(* CODESYS project XPlanarApplication143.library
   Placeholder: XPlanarApplication
   Version: 1.4.3
   Title: XPlanarApplication
   DefaultNamespace: XPlanarApplication
   Company: Beckhoff Automation LLC

Project tree, tasks and I/O mapping:
  libraries: SPT Base Types, * (Beckhoff Automation LLC); Tc2_Math, * (Beckhoff Automation GmbH); Tc2_Standard, * (Beckhoff Automation GmbH); Tc2_System, * (Beckhoff Automation GmbH); Tc2_Utilities, * (Beckhoff Automation GmbH); Tc3_EventLogger, * (Beckhoff Automation GmbH); Tc3_Mc3PlanarMotion, * (Beckhoff Automation GmbH); Tc3_Module, * (Beckhoff Automation GmbH); Tc3_Physics, * (Beckhoff Automation GmbH); Tc3_XPlanarUtility, * (Beckhoff Automation GmbH)
  Mover/
    DUTs/
      data type ST_CommandLog
      data type ST_MoveDynamics
      data type ST_MoverCommand
      data type ST_MoverHMI
      data type ST_MoverObjectInfos
    TaskClasses/
      function block FB_AddToGroup [ST]: Execute
      function block FB_Disable [ST]: Execute
      function block FB_Enable [ST]: Execute
      function block FB_EnterMovementArea [ST]: Execute, Update
      function block FB_Halt [ST]: Execute
      function block FB_JoinClosestTrack [ST]: Execute, Update
      function block FB_JoinTrack [ST]: Execute
      function block FB_LeaveMovementArea [ST]: Execute, Update
      function block FB_LeaveTrack [ST]: Execute
      function block FB_MoveA [ST]: Execute
      function block FB_MoveB [ST]: Execute
      function block FB_MoveToPosition [ST]: Execute
      function block FB_MoveZ [ST]: Execute
      function block FB_ResetMover [ST]: Execute
      function block FB_Rotate [ST]: Execute
      function block FB_RunExternalSetpointAbsoluteMode [ST]: Execute
      function block FB_RunExternalSetpointRelativeMode [ST]: Execute
      function block FB_SquareUp [ST]: Execute, Update
      function block FB_StopExternalSetpoint [ST]: Execute
      function block FB_TrackMove [ST]: Execute
      function block FB_TrackMoveXY [ST]: Execute
    function block FB_XPlanarMover [ST]: FreeMove, JoinClosestTrack, JoinTrack, LeaveTrack, Rotate, RunExternalSpAbsoluteMode, RunExternalSpRelativeMode, SendToStation, SquareUp, StopExternalSp, TiltA, TiltB, TrackMove, TrackMoveXY, VerticalMove, Movement, Rotation, Tilt, ActualPosition, AddToGroup, AtRotationPosition, CommandLog, Destination, Disable, Dynamics, Enable, EnterMovementArea, Gap, Halt, IdentifiedBTN, InStation, LeaveMovementArea, MoveCommand, MoverBTN, MoverIndex, MoverType, pm, Reset, RotationModulo, Status, Utility, CyclicLogic, Initialize
    interface I_MoveCommands: FreeMove, JoinClosestTrack, JoinTrack, LeaveTrack, Rotate, RunExternalSpAbsoluteMode, RunExternalSpRelativeMode, SendToStation, SquareUp, StopExternalSp, TiltA, TiltB, TrackMove, TrackMoveXY, VerticalMove
    interface I_MoveDynamics: Movement, Rotation, Tilt
    interface I_XPlanarMover: ActualPosition, AddToGroup, AtRotationPosition, CommandLog, CyclicLogic, Destination, Disable, Dynamics, Enable, EnterMovementArea, Gap, Halt, IdentifiedBTN, InStation, LeaveMovementArea, MoveCommand, MoverBTN, MoverIndex, MoverType, pm, Reset, RotationModulo, Status, Utility
  Part/
    Tasks/
      function block FB_AllowEnable [ST]: Execute
      function block FB_ForceDisable [ST]: Execute
      function block FB_Initialize [ST]: Execute
      function block FB_ResetPart [ST]: Execute
    function block FB_XPlanarPart [ST]: CyclicLogic, ForceDisable, Initialize, ObjectID, pm, Reset, SetAllowEnable, State
    interface I_XPlanarPart: ForceDisable, ObjectID, pm, Reset, SetAllowEnable, State
  Station/
    DUT/
      data type E_StationType
      data type E_XplanarStationState
      data type ST_StationHMI
      data type ST_XPlanarStationObjectInfos
    function block FB_MoverQueue [ST]: Clear, Count, Dequeue, Enqueue, FirstMover, LastMover, MoverIDs, Queue
    function block FB_XPlanarStationBase [ST]: AllowQueing, CanReleaseMover, CurrentMover, Error, Execute, HasMover, ID, MoverQueue, NextStation, NumMoversRequired, Position, Reset, Size, StationComplete, StationReady, StationType, TrackID, CyclicLogic, Name, WatchForMover
    interface I_XPlanarStation: AllowQueing, CanReleaseMover, CurrentMover, Execute, HasMover, ID, MoverQueue, Name, NextStation, NumMoversRequired, Position, Reset, Size, StationComplete, StationReady, StationType, TrackID
  Tile/
    DUT/
      data type ST_TileObjectInfos
      data type ST_TileTemperatures
    function block FB_XPlanarTile [ST]: Btn, CyclicLogic, DcLinkOk, Index, Initialize, PartIndex, PositionOnPart, Temperatures, TimeToShutdown, Update, Utility
    interface I_XPlanarTile: Btn, DcLinkOk, Index, PartIndex, PositionOnPart, Temperatures, TimeToShutdown, Update, Utility
  Track/
    DUT/
      data type E_TrackItemType
      data type ST_TrackDefinition
      data type ST_TrackItems
      data type ST_TrackStatus
    TaskClasses/
      function block FB_AddTrackToGroup [ST]: Execute
      function block FB_AppendLine [ST]: Execute
      function block FB_AppendPoint [ST]: Execute
      function block FB_BuildTrack [ST]: Execute, Update
      function block FB_ClearSegment [ST]: Execute
      function block FB_CloseLoop [ST]: Execute
      function block FB_DisableTrack [ST]: Execute
      function block FB_EnableTrack [ST]: Execute
      function block FB_SetEndAtTrack [ST]: Execute
      function block FB_SetStartFromTrack [ST]: Execute
      function block FB_TrackReset [ST]: Execute
    function block FB_XPlanarTrackSegment [ST]: AddToGroup, AppendLine, AppendPoint, Build, Clear, CloseLoop, Definition, Disable, Enable, GetTrackPositionAt, Index, IsStanding, MoverCount, MovingMoverCount, pm, Reset, SetEndAtTrack, SetStartFromTrack, Status, TrackLength, Utility, CyclicLogic
    interface I_XPlanarTrack: AddToGroup, AppendLine, AppendPoint, Build, Clear, CloseLoop, CyclicLogic, Definition, Disable, Enable, GetTrackPositionAt, Index, MoverCount, MovingMoverCount, pm, Reset, Status, TrackLength, Utility
  XPlanarComponent/
    TaskClasses/
      function block FB_EnableGroup [ST]: Execute
      function block FB_MoverIdentification [ST]: Execute, Update
      function block FB_MoverRedetection [ST]: Execute, MoverDetectionInfo, Update
      function block FB_ResetGroup [ST]: Execute
      function block FB_ResetXPlanar [ST]: Execute, Update
    function block FB_Component_XPlanar [ST]: Monitoring, CyclicLogic, Abort, AddMoversToGroup, AddTracksToGroup, DisableMovers, EnableGroup, EnableMovers, EnableTracks, IdentifyMovers, Initialize, MoverDetectionInfo, MoverRedetect, Reset, TileCount, TracksInitialized, Utility
  XPlanarResultClasses/
    function block FB_MoverTaskResult [ST]: Mover, Update, UpdateLog
    function block FB_PartTaskResult [ST]: Part
    function block FB_PlanarFeedbackResult [ST]: PlanarFeedback, Update
    function block FB_ResultBase [ST]: Aborted, BlockingObjectInfo, Busy, Done, Error, ErrorID, Result, TaskName
    function block FB_TrackTaskResult [ST]: Track
    interface I_PlanarTaskResult: Aborted, BlockingObjectInfo, Busy, Done, Error, ErrorID
  global variables ip
  00000000-0000-0000-0000-000000000000|LICENSE
  LICENSE
  global variables SystemParameters
  global variables XPlanar
  global variables XPlanarHMI
*)

// Mover/DUTs/ST_CommandLog
TYPE ST_CommandLog EXTENDS ST_MoverCommand :
	STRUCT
		Timestamp : STRING(24);
	END_STRUCT
END_TYPE

// Mover/DUTs/ST_MoveDynamics
TYPE ST_MoveDynamics :
STRUCT
	Velocity	: LREAL;
	Accel		: LREAL;
	Decel		: LREAL;
	Jerk		: LREAL;
END_STRUCT
END_TYPE

// Mover/DUTs/ST_MoverCommand
TYPE ST_MoverCommand :
	STRUCT
		Command : STRING;
		Vlocity : LREAL;
		Accel	: LREAL;
		Decel	: LREAL;
		Jerk	: LREAL;
	END_STRUCT
END_TYPE

// Mover/DUTs/ST_MoverHMI
TYPE ST_MoverHMI :
	STRUCT
		Enabled		   : BOOL;
		Error		   : BOOL;
		InStation	   : BOOL;
		ErrorID		   : UDINT;
		CurrentStation : STRING;
		CommandMode	   : STRING;
		LastCommand	   : STRING;
		EnableMover	   : BOOL;
		DisableMover   : BOOL;
		ResetMover	   : BOOL;
		HaltMover	   : BOOL;
	END_STRUCT
END_TYPE

// Mover/DUTs/ST_MoverObjectInfos
TYPE ST_MoverObjectInfos :
	STRUCT
		Width	 : DINT;
		Height	 : DINT;
		MoverBTN : STRING(13);
	END_STRUCT
END_TYPE

// Station/DUT/E_StationType
{attribute 'qualified_only'}
TYPE E_StationType : (
		Process		  := 0,
		DecisionPoint := 1,
		MultiMover	  := 2
	) UDINT;
END_TYPE

// Station/DUT/E_XplanarStationState
{attribute 'qualified_only'}
{attribute 'strict'}
{attribute 'to_string'}
TYPE E_XplanarStationState : (
		StationIdle := 0,
		ProcessMover,
		SquareUpMover,
		SendMoverAway,
		CycleComplete,
		SendQueue,
		StationError
	);
END_TYPE

// Station/DUT/ST_StationHMI
TYPE ST_StationHMI :
	STRUCT
		Error		   : BOOL;
		Reset		   : BOOL;
		StationReady   : BOOL;
		HasMover	   : BOOL;
		CurrentMoverID : STRING(13);
		CurrentState   : STRING;
	END_STRUCT
END_TYPE

// Station/DUT/ST_XPlanarStationObjectInfos
TYPE ST_XPlanarStationObjectInfos :
	STRUCT
		X	   : DINT;
		Y	   : DINT;
		Width  : DINT;
		Height : DINT;
	END_STRUCT
END_TYPE

// Tile/DUT/ST_TileObjectInfos
TYPE ST_TileObjectInfos :
	STRUCT
		X	   : DINT;
		Y	   : DINT;
		Width  : DINT;
		Height : DINT;
	END_STRUCT
END_TYPE

// Tile/DUT/ST_TileTemperatures
TYPE ST_TileTemperatures :
	STRUCT
		Center : LREAL;
		East   : LREAL;
		West   : LREAL;
		North  : LREAL;
		South  : LREAL;
	END_STRUCT
END_TYPE

// Track/DUT/E_TrackItemType
TYPE E_TrackItemType :
(
	Point := 0,
	Line,
	Circle
);
END_TYPE

// Track/DUT/ST_TrackDefinition
TYPE ST_TrackDefinition :
	STRUCT
		StartFromTrackID : UDINT;
		EndAtTrackID	 : UDINT;
		CloseLoop		 : BOOL;
		Items			 : ARRAY[1..SystemParameters.MAX_OBJECTS_PER_TRACK] OF ST_TrackItems;
	END_STRUCT
END_TYPE

// Track/DUT/ST_TrackItems
TYPE ST_TrackItems :
STRUCT
	ItemType		: E_TrackItemType;
	StartPoint		: PositionXYC;
	EndPoint		: PositionXYC;
	CenterPoint		: PositionXY;
	CircleClockwise : BOOL;
END_STRUCT
END_TYPE

// Track/DUT/ST_TrackStatus
TYPE ST_TrackStatus :
	STRUCT
		State			 : MC_PLANAR_STATE;
		OperationMode	 : MC_PLANAR_TRACK_OPERATION_MODE;
		MoverCount		 : UDINT;
		CalculatedLength : LREAL;
	END_STRUCT
END_TYPE

// ip
{attribute 'qualified_only'}
VAR_GLOBAL
	Movers	 : ARRAY[0..SystemParameters.MOVER_COUNT] OF I_XPlanarMover;
	Tracks	 : ARRAY[0..SystemParameters.TRACK_COUNT] OF I_XPlanarTrack;
	Stations : ARRAY[0..SystemParameters.STATION_COUNT] OF I_XPlanarStation;
END_VAR

// SystemParameters
{attribute 'qualified_only'}
VAR_GLOBAL CONSTANT
	EnableCommandTracing  : BOOL  := FALSE; //Enables mover command trace logging
	AssumedMoverSize	  : LREAL := 50;
	MAX_LOG_COUNT		  : UINT  := 20; //Size of command mover log
	MOVER_COUNT			  : UINT  := 1;	 //Total number of movers configured in the system
	TRACK_COUNT			  : UINT  := 1;	 //Total number of track segments in the system
	MAX_OBJECTS_PER_TRACK : UINT  := 20; //Maximum number of points or lines defined in a single track segment
	STATION_COUNT		  : UINT  := 3;	 //Total number of stations in the system
	MaxMoversPerStation	  : UDINT := 4;	 //Max number of movers allowed to queue in a station 
	TileDiagUpdate		  : LREAL := 0;	 //Tile Diagnostic data update rate in seconds.  Set to 0 to disable
END_VAR

// XPlanar
{attribute 'qualified_only'}
VAR_GLOBAL
	Environment		   : Tc3_MC3PlanarMotion.MC_PlanarEnvironment;
	EnvironmentTcIo	   : Tc3_XPlanarUtility.FB_TcIoXPlanarEnvironment;
	Group			   : Tc3_MC3PlanarMotion.MC_PlanarGroup;
	Parts			   : ARRAY[1..Param_TcIoXPlanarEnvironment.MaxParts] OF FB_XPlanarPart;
	Tiles			   : ARRAY[1..Param_TcIoXPlanarEnvironment.MaxTiles] OF FB_XPlanarTile;
	OperationMode	   : XPlanarOperationMode;
	RotationMultiplier : LREAL := 120.0;
	XPUCount		   : UINT;
	PartCount		   : UINT;
	TrackCount		   : UINT;
	MoverCount		   : UINT;
	TileCount		   : UINT;
END_VAR

// XPlanarHMI
{attribute 'qualified_only'}
VAR_GLOBAL
	MoverObjects	: ARRAY[1..SystemParameters.MOVER_COUNT] OF ST_MoverObjectInfos;
	MoverPositions	: ARRAY[1..SystemParameters.MOVER_COUNT] OF MoverVector;
	TileObjects		: ARRAY[1..Param_TcIoXPlanarEnvironment.MaxTiles] OF ST_TileObjectInfos;
	StationObjects	: ARRAY[1..SystemParameters.STATION_COUNT] OF ST_XPlanarStationObjectInfos;
END_VAR

// Mover/TaskClasses/FB_AddToGroup
FUNCTION_BLOCK FB_AddToGroup EXTENDS FB_MoverTaskResult
VAR
END_VAR

METHOD Execute : I_PlanarTaskResult
VAR_INPUT
	Group : REFERENCE TO MC_PlanarGroup;
END_VAR
IF NOT HasRun THEN
	_Done	 := FALSE;
	_Error	 := FALSE;
	_Busy	 := FALSE;
	_ErrorID := 0;
	ipMover.pm.AddToGroup(_PlanarFb, Group);

	//Update mover command log				
	LogEntry.Command := CONCAT('AddMoverToGroup ', TO_STRING(Group.MCTOPLC_STD.GroupOID));
	LogEntry.Accel	 := 0;
	LogEntry.Decel	 := 0;
	LogEntry.Jerk	 := 0;
	LogEntry.Vlocity := 0;
	UpdateLog();
	HasRun := TRUE;
END_IF

Execute := THIS^;

//Heartbeat that the method is active
ExecuteWatchdog := ExecuteWatchdog + 1;
END_METHOD

END_FUNCTION_BLOCK

// XPlanarResultClasses/FB_MoverTaskResult
{attribute 'no_explicit_call' := 'do not call this POU directly'}
FUNCTION_BLOCK FB_MoverTaskResult EXTENDS FB_PlanarFeedbackResult
VAR
	ipMover : I_XPlanarMover;

	//CmdLog		   : REFERENCE TO ARRAY[0..SystemParameters.MAX_LOG_COUNT] OF ST_CommandLog;
	GetTime		   : GETSYSTEMTIME;
	SysTime		   : T_FILETIME;
	LogEntry	   : ST_MoverCommand;
	ActualPosition : MoverVector;
	RT_ADSWarn	   : R_Trig;
	MoverStr	   : STRING;
END_VAR

PROPERTY Mover : I_XPlanarMover
SET
ipMover := Mover;
END_SET
END_PROPERTY

METHOD Update
ActualPosition := ipMover.ActualPosition;
SUPER^.Update();
RT_ADSWarn(CLK := _PlanarFb.Error);
IF RT_ADSWarn.Q THEN
	MoverStr := CONCAT('Mover ', TO_STRING(ipMover.MoverIndex));
	LogEntry.Command := CONCAT(CONCAT(MoverStr, ' : %s'), CONCAT(LogEntry.Command, CONCAT('Error ', TO_STRING(_PlanarFb.ErrorId))));
	UpdateLog();
END_IF
END_METHOD

METHOD UpdateLog
VAR_INST
	i : UINT;
END_VAR
IF SystemParameters.MAX_LOG_COUNT > 0 THEN
	FOR i := SystemParameters.MAX_LOG_COUNT - 1 TO 1 BY -1 DO
		IF i < SystemParameters.MAX_LOG_COUNT THEN
			ipMover.CommandLog[i + 1] := ipMover.CommandLog[i];
		END_IF
	END_FOR

	ipMover.CommandLog[1] := ipMover.CommandLog[0];
	GetTime(timeLoDW => SysTime.dwLowDateTime, timeHiDW => SysTime.dwHighDateTime);
	ipMover.CommandLog[0].Timestamp := SYSTEMTIME_TO_STRING(FILETIME_TO_SYSTEMTIME(SysTime));
	ipMover.CommandLog[0].Command	:= LogEntry.Command;
	ipMover.CommandLog[0].Accel		:= LogEntry.Accel;
	ipMover.CommandLog[0].Decel		:= LogEntry.Decel;
	ipMover.CommandLog[0].Jerk		:= LogEntry.Jerk;
	ipMover.CommandLog[0].Vlocity	:= LogEntry.Vlocity;
END_IF
END_METHOD

END_FUNCTION_BLOCK

// XPlanarResultClasses/FB_PlanarFeedbackResult
{attribute 'no_assign_warning'}
{attribute 'no_explicit_call' := 'do not call this POU directly'}
FUNCTION_BLOCK FB_PlanarFeedbackResult EXTENDS FB_ResultBase
VAR
	_PlanarFb		: MC_PlanarFeedback;
	HasRun			: BOOL;
	ExecuteWatchdog : UDINT;
	TaskState		: UDINT;
END_VAR

{attribute 'suppress_wrn_C0410'}
PROPERTY PlanarFeedback : REFERENCE TO MC_PlanarFeedback
GET
PlanarFeedback ref= _PlanarFb;
END_GET
END_PROPERTY

METHOD Update
VAR_INST
	WatchdogCheck : UDINT;
END_VAR
//Update Command Feedback Status
_PlanarFb.Update();

//Update Interface based on Command Feedback status
_Aborted			:= _PlanarFb.Aborted;
_Busy				:= _PlanarFb.Active OR _PlanarFb.Busy;
_Done				:= _PlanarFb.Done;
_Error				:= _PlanarFb.Error;
_ErrorID			:= _PlanarFb.ErrorId;
_BlockingObjectInfo := _PlanarFb.objectInfo;

//Heartbeat to know execute is active
IF ExecuteWatchdog <> WatchdogCheck THEN
	WatchdogCheck := ExecuteWatchdog;
ELSE
	HasRun			:= FALSE;
	ExecuteWatchdog := 0;
END_IF
END_METHOD

END_FUNCTION_BLOCK

// XPlanarResultClasses/FB_ResultBase
{attribute 'no_explicit_call' := 'do not call this POU directly'}
FUNCTION_BLOCK FB_ResultBase EXTENDS FB_BaseFB IMPLEMENTS I_PlanarTaskResult
VAR
	_TaskName			: STRING;
	_Done				: BOOL;
	_Aborted			: BOOL;
	_BlockingObjectInfo : PlanarObjectInfo;
END_VAR

{attribute 'monitoring' := 'call'}
PROPERTY Aborted : BOOL
GET
Aborted := _Aborted;
END_GET
SET
_Aborted := Aborted;
END_SET
END_PROPERTY

{attribute 'suppress_wrn_C0410'}
PROPERTY BlockingObjectInfo : REFERENCE TO Tc3_Mc3PlanarMotion.PlanarObjectInfo
GET
BlockingObjectInfo ref= _BlockingObjectInfo;
END_GET
END_PROPERTY

{attribute 'monitoring' := 'call'}
PROPERTY Busy : BOOL
GET
Busy := _Busy;
END_GET
SET
_Busy := Busy;
END_SET
END_PROPERTY

{attribute 'monitoring' := 'call'}
PROPERTY Done : BOOL
GET
Done := _Done;
END_GET
SET
_Done := Done;
END_SET
END_PROPERTY

{attribute 'monitoring' := 'call'}
PROPERTY Error : BOOL
GET
Error := _Error;
END_GET
SET
_Error := Error;
END_SET
END_PROPERTY

{attribute 'monitoring' := 'call'}
PROPERTY ErrorID : UDINT
GET
ErrorID := _ErrorID;
END_GET
SET
_ErrorID := ErrorID;
END_SET
END_PROPERTY

PROPERTY Result : I_PlanarTaskResult
GET
Result := THIS^;
END_GET
END_PROPERTY

PROPERTY TaskName : STRING
GET
TaskName := _TaskName;
END_GET
SET
_TaskName := TaskName;
END_SET
END_PROPERTY

END_FUNCTION_BLOCK

// XPlanarResultClasses/I_PlanarTaskResult
INTERFACE I_PlanarTaskResult

{attribute 'monitoring' := 'call'}
PROPERTY Aborted : BOOL
GET
END_GET
END_PROPERTY

{attribute 'suppress_wrn_C0410'}
PROPERTY BlockingObjectInfo : REFERENCE TO PlanarObjectInfo
GET
END_GET
END_PROPERTY

{attribute 'monitoring' := 'call'}
PROPERTY Busy : BOOL
GET
END_GET
END_PROPERTY

{attribute 'monitoring' := 'call'}
PROPERTY Done : BOOL
GET
END_GET
END_PROPERTY

{attribute 'monitoring' := 'call'}
PROPERTY Error : BOOL
GET
END_GET
END_PROPERTY

{attribute 'monitoring' := 'call'}
PROPERTY ErrorID : UDINT
GET
END_GET
END_PROPERTY

END_INTERFACE

// Mover/I_XPlanarMover
INTERFACE I_XPlanarMover EXTENDS I_BaseFb

{attribute 'suppress_wrn_C0410'}
PROPERTY ActualPosition : REFERENCE TO MoverVector
GET
END_GET
END_PROPERTY

METHOD AddToGroup : I_PlanarTaskResult
VAR_INPUT
	PlanarGroup : REFERENCE TO MC_PlanarGroup;
END_VAR
END_METHOD

PROPERTY AtRotationPosition : BOOL
GET
END_GET
END_PROPERTY

{attribute 'suppress_wrn_C0410'}
PROPERTY CommandLog : REFERENCE TO ARRAY [0..SystemParameters.MAX_LOG_COUNT] of ST_CommandLog
GET
END_GET
END_PROPERTY

{attribute 'hide'}
METHOD CyclicLogic
END_METHOD

PROPERTY Destination : I_XPlanarStation
GET
END_GET
SET
END_SET
END_PROPERTY

METHOD Disable : I_PlanarTaskResult
END_METHOD

PROPERTY Dynamics : I_MoveDynamics
GET
END_GET
END_PROPERTY

METHOD Enable : I_PlanarTaskResult
END_METHOD

METHOD EnterMovementArea : I_PlanarTaskResult
VAR_INPUT
	PartId		: OTCID;
	PositionX	: LREAL;
	PositionY	: LREAL;
END_VAR
END_METHOD

PROPERTY Gap : LREAL
GET
END_GET
SET
END_SET
END_PROPERTY

METHOD Halt : I_PlanarTaskResult
END_METHOD

PROPERTY IdentifiedBTN : STRING
GET
END_GET
SET
END_SET
END_PROPERTY

PROPERTY InStation : BOOL
GET
END_GET
SET
END_SET
END_PROPERTY

METHOD LeaveMovementArea : I_PlanarTaskResult
END_METHOD

PROPERTY MoveCommand : I_MoveCommands
GET
END_GET
END_PROPERTY

PROPERTY MoverBTN : STRING
GET
END_GET
END_PROPERTY

PROPERTY MoverIndex : UDINT
GET
END_GET
SET
END_SET
END_PROPERTY

PROPERTY MoverType : XplanarMoverType
GET
END_GET
SET
END_SET
END_PROPERTY

{attribute 'suppress_wrn_C0410'}
PROPERTY pm : REFERENCE TO MC_PlanarMover
GET
END_GET
END_PROPERTY

//! @summary Clears error flags and error IDs for this component
{attribute 'TcRpcEnable'}
METHOD PUBLIC Reset : I_PlanarTaskResult
END_METHOD

PROPERTY RotationModulo : LREAL
GET
END_GET
END_PROPERTY

{attribute 'suppress_wrn_C0410'}
PROPERTY Status : REFERENCE TO CDT_MCTOPLC_PLANAR_MOVER_STD
GET
END_GET
END_PROPERTY

PROPERTY Utility : I_TcIoXPlanarMover
GET
END_GET
SET
END_SET
END_PROPERTY

END_INTERFACE

// Station/I_XPlanarStation
INTERFACE I_XPlanarStation EXTENDS I_BaseFb

PROPERTY AllowQueing : BOOL
GET
END_GET
SET
END_SET
END_PROPERTY

PROPERTY CanReleaseMover : BOOL
SET
END_SET
END_PROPERTY

PROPERTY CurrentMover : I_XPlanarMover
GET
END_GET
END_PROPERTY

METHOD Execute
END_METHOD

PROPERTY HasMover : BOOL
GET
END_GET
SET
END_SET
END_PROPERTY

PROPERTY ID : UDINT
GET
END_GET
SET
END_SET
END_PROPERTY

{attribute 'suppress_wrn_C0410'}
PROPERTY MoverQueue : REFERENCE TO FB_MoverQueue
GET
END_GET
END_PROPERTY

PROPERTY Name : STRING
GET
END_GET
SET
END_SET
END_PROPERTY

PROPERTY NextStation : I_XPlanarStation
GET
END_GET
SET
END_SET
END_PROPERTY

PROPERTY NumMoversRequired : UDINT
GET
END_GET
SET
END_SET
END_PROPERTY

{attribute 'suppress_wrn_C0410'}
PROPERTY Position : REFERENCE TO PositionXYC
GET
END_GET
END_PROPERTY

METHOD Reset : BOOL
END_METHOD

{attribute 'suppress_wrn_C0410'}
PROPERTY Size : REFERENCE TO Position2D_LREAL
GET
END_GET
END_PROPERTY

PROPERTY StationComplete : BOOL
SET
END_SET
END_PROPERTY

PROPERTY StationReady : BOOL
GET
END_GET
END_PROPERTY

PROPERTY StationType : E_StationType
GET
END_GET
SET
END_SET
END_PROPERTY

PROPERTY TrackID : UDINT
GET
END_GET
SET
END_SET
END_PROPERTY

END_INTERFACE

// Station/FB_MoverQueue
//=============================================================================
//	FB_MoverQueue
//=============================================================================
//
//	FIFO Queue for use by stations
//
//-----------------------------------------------------------------------------

FUNCTION_BLOCK FB_MoverQueue
VAR
	MoversInQueue : UDINT := 0;
	ipMovers	  : ARRAY[1..SystemParameters.MaxMoversPerStation] OF I_XPlanarMover;
END_VAR

//=============================================================================
//	Method Clear()
//=============================================================================
//
//	Brute force reset of buffer
//
//-----------------------------------------------------------------------------
METHOD Clear : BOOL
MEMSET(ADR(ipMovers), 0, SIZEOF(ipMovers));
MoversInQueue := 0;
Clear		  := TRUE;
END_METHOD

PROPERTY Count : UDINT
GET
VAR
	i	 : UDINT;
	temp : UDINT;
END_VAR
Count := MoversInQueue;
END_GET
END_PROPERTY

METHOD Dequeue : BOOL
IF MoversInQueue > 0 THEN
	ipMovers[1].InStation := FALSE;
	MEMSET(ADR(ipMovers[1]), 0, SIZEOF(ipMovers[1]));
	MoversInQueue := MoversInQueue - 1;
	IF MoversInQueue > 0 THEN
		MEMMOVE(ADR(ipMovers[1]), ADR(ipMovers[2]), SIZEOF(ipMovers[2]) * MoversInQueue);
		MEMSET(ADR(ipMovers[MoversInQueue + 1]), 0, (SIZEOF(ipMovers[1]) * (SystemParameters.MaxMoversPerStation - MoversInQueue)));
	END_IF

	Dequeue := TRUE;
END_IF
END_METHOD

METHOD Enqueue : BOOL
VAR_INPUT
	ipMover : I_XPlanarMover;
END_VAR
IF MoversInQueue < SystemParameters.MaxMoversPerStation THEN
	MoversInQueue			:= MoversInQueue + 1;
	ipMover.InStation		:= TRUE;
	ipMovers[MoversInQueue] := ipMover;
	Enqueue					:= TRUE;
END_IF
END_METHOD

PROPERTY FirstMover : I_XPlanarMover
GET
IF MoversInQueue > 0 THEN
	FirstMover := ipMovers[1];
END_IF
END_GET
END_PROPERTY

PROPERTY LastMover : I_XPlanarMover
GET
IF MoversInQueue > 0 THEN
	LastMover := ipMovers[MoversInQueue];
END_IF
END_GET
END_PROPERTY

PROPERTY MoverIDs : ARRAY[1..SystemParameters.MaxMoversPerStation] OF UDINT
GET
VAR
	i : UDINT;
END_VAR
FOR i := 1 TO MoversInQueue DO
	IF ipMovers[i] <> 0 THEN
		MoverIDs[i] := ipMovers[i].MoverIndex;
	END_IF
END_FOR
END_GET
END_PROPERTY

{attribute 'suppress_wrn_C0410'}
PROPERTY Queue : REFERENCE TO ARRAY[1..SystemParameters.MaxMoversPerStation] OF I_XPlanarMover;
GET
VAR
	i : UDINT;
END_VAR
Queue ref= ipMovers;
END_GET
END_PROPERTY

END_FUNCTION_BLOCK

// Mover/I_MoveDynamics
INTERFACE I_MoveDynamics EXTENDS __SYSTEM.IQueryInterface

{attribute 'suppress_wrn_C0410'}
PROPERTY Movement : REFERENCE TO ST_MoveDynamics
GET
END_GET
END_PROPERTY

{attribute 'suppress_wrn_C0410'}
PROPERTY Rotation : REFERENCE TO ST_MoveDynamics
GET
END_GET
END_PROPERTY

{attribute 'suppress_wrn_C0410'}
PROPERTY Tilt : REFERENCE TO ST_MoveDynamics
GET
END_GET
END_PROPERTY

END_INTERFACE

// Mover/I_MoveCommands
INTERFACE I_MoveCommands EXTENDS __SYSTEM.IQueryInterface

METHOD FreeMove : I_PlanarTaskResult
VAR_INPUT
	XPosition : LREAL;
	YPosition : LREAL;
END_VAR
END_METHOD

{attribute 'TcRpcEnable'}
METHOD JoinClosestTrack : I_PlanarTaskResult
VAR_INPUT
	UseOrientation : BOOL;
END_VAR
END_METHOD

{attribute 'TcRpcEnable'}
METHOD JoinTrack : I_PlanarTaskResult
VAR_INPUT
	ipTrack		   : I_XPlanarTrack;
	UseOrientation : BOOL;
END_VAR
END_METHOD

{attribute 'TcRpcEnable'}
METHOD LeaveTrack : I_PlanarTaskResult
VAR_INPUT
	DestinationX   : LREAL;
	DestinationY   : LREAL;
	UseOrientation : BOOL;
END_VAR
END_METHOD

{attribute 'TcRpcEnable'}
METHOD Rotate : I_PlanarTaskResult
VAR_INPUT
	Position		: LREAL;
	AdditionalTurns : DINT;
END_VAR
END_METHOD

METHOD RunExternalSpAbsoluteMode : I_PlanarTaskResult
VAR_INPUT
	Position	 : MoverVector;
	Velocity	 : MoverVector;
	Acceleration : MoverVector;
END_VAR
END_METHOD

METHOD RunExternalSpRelativeMode : I_PlanarTaskResult
VAR_INPUT
	Position	 : MoverVector;
	Velocity	 : MoverVector;
	Acceleration : MoverVector;
END_VAR
END_METHOD

{attribute 'TcRpcEnable'}
METHOD SendToStation : I_PlanarTaskResult
VAR_INPUT
	Destination : I_XPlanarStation;
END_VAR
END_METHOD

{attribute 'TcRpcEnable'}
METHOD SquareUp : I_PlanarTaskResult
END_METHOD

METHOD StopExternalSp : I_PlanarTaskResult
END_METHOD

METHOD TiltA : I_PlanarTaskResult
VAR_INPUT
	Position : LREAL;
END_VAR
END_METHOD

METHOD TiltB : I_PlanarTaskResult
VAR_INPUT
	Position : LREAL;
END_VAR
END_METHOD

{attribute 'TcRpcEnable'}
METHOD TrackMove : I_PlanarTaskResult
VAR_INPUT
	Position : LREAL;
	Gap		  : LREAL;
	Track	  : I_XPlanarTrack;
	Direction : Tc3_Mc3PlanarMotion.MC_DIRECTION;
END_VAR
END_METHOD

{attribute 'TcRpcEnable'}
METHOD TrackMoveXY : I_PlanarTaskResult
VAR_INPUT
	XPosition : LREAL;
	YPosition : LREAL;
	Gap		  : LREAL;
	Track	  : I_XPlanarTrack;
	Direction : Tc3_Mc3PlanarMotion.MC_DIRECTION;
END_VAR
END_METHOD

{attribute 'TcRpcEnable'}
METHOD VerticalMove : I_PlanarTaskResult
VAR_INPUT
	Position : LREAL;
END_VAR
END_METHOD

END_INTERFACE

// Track/I_XPlanarTrack
INTERFACE I_XPlanarTrack EXTENDS I_BaseFb

METHOD AddToGroup : I_PlanarTaskResult
VAR_INPUT
	PlanarGroup : REFERENCE TO MC_PlanarGroup;
END_VAR
END_METHOD

METHOD AppendLine : I_PlanarTaskResult
VAR_INPUT
	StartPointX : LREAL;
	StartPointY : LREAL;
	EndPointX	: LREAL;
	EndPointY	: LREAL;
END_VAR
END_METHOD

METHOD AppendPoint : I_PlanarTaskResult
VAR_INPUT
	XPoint : LREAL;
	YPoint : LREAL;
END_VAR
END_METHOD

METHOD Build : I_PlanarTaskResult
END_METHOD

METHOD Clear : I_PlanarTaskResult
END_METHOD

METHOD CloseLoop : I_PlanarTaskResult
END_METHOD

{attribute 'hide'}
METHOD CyclicLogic
END_METHOD

{attribute 'suppress_wrn_C0410'}
PROPERTY Definition : REFERENCE TO ST_TrackDefinition
GET
END_GET
END_PROPERTY

METHOD Disable : I_PlanarTaskResult
END_METHOD

{attribute 'TcRpcEnable'}
METHOD Enable : I_PlanarTaskResult
END_METHOD

METHOD GetTrackPositionAt : LREAL;
VAR_IN_OUT
	Position : PositionXYC;
END_VAR
END_METHOD

PROPERTY Index : UDINT
GET
END_GET
SET
END_SET
END_PROPERTY

PROPERTY MoverCount : UDINT
GET
END_GET
END_PROPERTY

PROPERTY MovingMoverCount : UDINT
GET
END_GET
END_PROPERTY

{attribute 'suppress_wrn_C0410'}
PROPERTY pm : REFERENCE TO MC_PlanarTrack
GET
END_GET
END_PROPERTY

METHOD Reset : I_PlanarTaskResult
VAR_INPUT
END_VAR
END_METHOD

{attribute 'suppress_wrn_C0410'}
PROPERTY Status : REFERENCE TO CDT_MCTOPLC_PLANAR_TRACK
GET
END_GET
END_PROPERTY

PROPERTY TrackLength : LREAL
GET
END_GET
END_PROPERTY

PROPERTY Utility : I_McPlanarTrack
GET
END_GET
END_PROPERTY

END_INTERFACE

// Mover/TaskClasses/FB_Disable
FUNCTION_BLOCK FB_Disable EXTENDS FB_MoverTaskResult
VAR
END_VAR

METHOD Execute : I_PlanarTaskResult
VAR_INPUT
END_VAR
IF NOT HasRun AND ipMover.Status.State <> MC_Planar_State.Disabled THEN
	_Done	 := FALSE;
	_Error	 := FALSE;
	_Busy	 := FALSE;
	_ErrorID := 0;
	ipMover.pm.Disable(_PlanarFb);

	//Update mover command log				
	LogEntry.Command := 'DisableMover';
	LogEntry.Accel	 := 0;
	LogEntry.Decel	 := 0;
	LogEntry.Jerk	 := 0;
	LogEntry.Vlocity := 0;
	UpdateLog();
	HasRun := TRUE;
END_IF

Execute := THIS^;

//Heartbeat that the method is active
ExecuteWatchdog := ExecuteWatchdog + 1;
END_METHOD

END_FUNCTION_BLOCK

// Mover/TaskClasses/FB_Enable
FUNCTION_BLOCK FB_Enable EXTENDS FB_MoverTaskResult
VAR
END_VAR

METHOD Execute : I_PlanarTaskResult
IF NOT HasRun AND ipMover.Status.State = MC_Planar_State.Disabled THEN
	_Done	 := FALSE;
	_Error	 := FALSE;
	_Busy	 := FALSE;
	_ErrorID := 0;
	ipMover.pm.Enable(_PlanarFb);

	//Update mover command log				
	LogEntry.Command := 'EnableMover';
	LogEntry.Accel	 := 0;
	LogEntry.Decel	 := 0;
	LogEntry.Jerk	 := 0;
	LogEntry.Vlocity := 0;
	UpdateLog();
	HasRun := TRUE;
END_IF

Execute := THIS^;

//Heartbeat that the method is active
ExecuteWatchdog := ExecuteWatchdog + 1;
END_METHOD

END_FUNCTION_BLOCK

// Mover/TaskClasses/FB_EnterMovementArea
FUNCTION_BLOCK FB_EnterMovementArea EXTENDS FB_MoverTaskResult
VAR
	MovementAreaParameters : EnterOrLeaveMovementAreaParameters;
	EnterMvmtArea		   : BOOL;
END_VAR

METHOD Execute : I_PlanarTaskResult
VAR_INPUT
	PartId		: OTCID;
	PositionX	: LREAL;
	PositionY	: LREAL;
END_VAR
IF NOT HasRun THEN
	_Done								   := FALSE;
	_Error								   := FALSE;
	_Busy								   := FALSE;
	_ErrorID							   := 0;
	MovementAreaParameters.MovementAreaOID := PartId;
	MovementAreaParameters.Positions.x	   := PositionX;
	MovementAreaParameters.Positions.y	   := PositionY;
	EnterMvmtArea						   := TRUE;
	HasRun								   := TRUE;

	//Update mover command log				
	LogEntry.Command := CONCAT('Add To Movement Area', TO_STRING(PartId));
	UpdateLog();
END_IF

Execute := THIS^;

//Heartbeat that the method is active
ExecuteWatchdog := ExecuteWatchdog + 1;
END_METHOD

METHOD Update
VAR_INST
	WatchdogCheck : UDINT;
END_VAR
//State logic for the task
CASE TaskState OF
	0: // Init
		_Busy := FALSE;
		IF EnterMvmtArea THEN
			_Done		  := FALSE;
			_Error		  := FALSE;
			_ErrorID	  := 0;
			_Busy		  := TRUE;
			EnterMvmtArea := FALSE;
			TaskState	  := TaskState + 10;
		END_IF

	10: //Check input parameters
		IF MovementAreaParameters.MovementAreaOID = 0 OR MovementAreaParameters.Positions.x = 0 OR MovementAreaParameters.Positions.x = 0 THEN
			_Error	  := TRUE;
			_ErrorID  := 9999; //Invalid Entry
			TaskState := 0;
		ELSE
			TaskState := TaskState + 10;
		END_IF

	20: //Set Mover Movement Area
		IF ipMover.Utility.SetMovementArea(MovementAreaParameters) THEN
			TaskState := TaskState + 10;
		END_IF

	30:
		IF SUCCEEDED(MovementAreaParameters.Result) THEN
			_Done	  := TRUE;
			TaskState := 0;
		ELSIF FAILED(MovementAreaParameters.Result) THEN
			_Error	  := TRUE;
			_ErrorID  := TO_UDINT(MovementAreaParameters.Result);
			TaskState := 0;
		END_IF
END_CASE

RT_ADSWarn(CLK := _Error);
IF RT_ADSWarn.Q THEN
	ADSLOGSTR(ADSLOG_MSGTYPE_WARN, CONCAT('Mover ', ipMover.MoverBTN), CONCAT(_TaskName, CONCAT('Error ', TO_STRING(_ErrorId))));
END_IF

IF ExecuteWatchdog <> WatchdogCheck THEN
	WatchdogCheck := ExecuteWatchdog;
ELSE
	HasRun			:= FALSE;
	ExecuteWatchdog := 0;
END_IF
END_METHOD

END_FUNCTION_BLOCK

// Mover/TaskClasses/FB_Halt
FUNCTION_BLOCK FB_Halt EXTENDS FB_MoverTaskResult
VAR
	BusyStatus : MoverBusy;
END_VAR

METHOD Execute : I_PlanarTaskResult
VAR_INPUT
	Dynamics : REFERENCE TO DynamicConstraint_Coordinates;
END_VAR
BusyStatus := ipMover.Status.Busy;
IF NOT HasRun AND BusyStatus.busyMover THEN
	_Done	 := FALSE;
	_Error	 := FALSE;
	_Busy	 := FALSE;
	_ErrorID := 0;
	ipMover.pm.Halt(_PlanarFb, Dynamics);

	//Update mover command log				
	LogEntry.Command := 'HaltMover';
	UpdateLog();
	HasRun := TRUE;
END_IF

Execute := THIS^;

//Heartbeat that the method is active
ExecuteWatchdog := ExecuteWatchdog + 1;
END_METHOD

END_FUNCTION_BLOCK

// Mover/TaskClasses/FB_JoinClosestTrack
{attribute 'no_assign_warning'}
FUNCTION_BLOCK FB_JoinClosestTrack EXTENDS FB_MoverTaskResult
VAR
	JoinTrackOptions	 : ST_JoinTrackOptions;
	TrackJoinDistances	 : ARRAY[1..SystemParameters.TRACK_COUNT] OF LREAL;
	_UseOrientation		 : BOOL;
	_MoveDynamics		 : DynamicConstraint_PathXYZ;
	i					 : UINT;
	MoverSetPosition	 : MoverVector;
	MoverCurrentPosition : PositionXYC;
	MoverJoinPosition	 :  ARRAY[1..SystemParameters.TRACK_COUNT] OF PositionXYC;
	MoverArcPosition	 :  ARRAY[1..SystemParameters.TRACK_COUNT] OF LREAL;
	ShortestDistance	 : LREAL;
	TrackToJoin			 : UINT;
	Join				 : BOOL;
END_VAR

METHOD Execute : I_PlanarTaskResult
VAR_INPUT
	UseOrientation : BOOL;
	MoveDynamics   : DynamicConstraint_PathXYZ;
END_VAR
IF NOT HasRun AND (ipMover.Status.CommandMode <> MC_Planar_Mover_Command_Mode.OnTrack) THEN
	_Done			:= FALSE;
	_Error			:= FALSE;
	_Busy			:= FALSE;
	_ErrorID		:= 0;
	_UseOrientation := UseOrientation;
	_MoveDynamics	:= MoveDynamics;
	Join			:= TRUE;
	HasRun			:= TRUE;
END_IF

Execute := THIS^;

//Heartbeat that the method is active
ExecuteWatchdog := ExecuteWatchdog + 1;
END_METHOD

METHOD Update
VAR_INST
	WatchdogCheck : UDINT;
END_VAR
//***Overwriting the update method because this task contains a state machine that must be monitored cyclically.***
_PlanarFb.Update();

//State logic for the task
CASE TaskState OF
	0: // Init
		_Busy := FALSE;
		IF Join THEN
			_Done			 := FALSE;
			_Error			 := FALSE;
			_ErrorID		 := 0;
			_Busy			 := TRUE;
			Join			 := FALSE;
			ShortestDistance := 0;
			TaskState		 := TaskState + 10;
		END_IF

	10: //Resolve Mover Position
		MoverSetPosition	   := ipMover.pm.MCTOPLC.SET.SetPos;
		MoverCurrentPosition.x := MoverSetPosition.x;
		MoverCurrentPosition.y := MoverSetPosition.y;
		MoverCurrentPosition.c := MoverSetPosition.c;
		TaskState			   := TaskState + 10;

	20: //Calculate distance from tracks
		FOR i := 1 TO SystemParameters.TRACK_COUNT DO
			//Get arc position based on mover position
			MoverArcPosition[i] := ip.Tracks[i].GetTrackPositionAt(MoverCurrentPosition);

			//Get Position based on arc position
			ip.Tracks[i].pm.GetPositionAt(MoverArcPosition[i], MoverJoinPosition[i]);

			//Save position delta
			TrackJoinDistances[i] := ABS(MoverJoinPosition[i].x - MoverCurrentPosition.x) + ABS(MoverJoinPosition[i].y - MoverCurrentPosition.y);
		END_FOR

		TaskState := TaskState + 10;

	30: //Find Closest Track
		FOR i := 1 TO SystemParameters.TRACK_COUNT DO
			IF ShortestDistance = 0 OR TrackJoinDistances[i] < ShortestDistance THEN
				ShortestDistance := TrackJoinDistances[i];
				TrackToJoin		 := i;
			END_IF
		END_FOR

		TaskState := TaskState + 10;

	40: //Join the closest track
		IF TrackToJoin > 0 THEN
			JoinTrackOptions.useOrientation := _UseOrientation;
			ipMover.pm.JoinTrack(_PlanarFb,
								 ip.Tracks[TrackToJoin].pm,
								 _MoveDynamics,
								 JoinTrackOptions);
	
			//Update mover command log				
			LogEntry.Command := CONCAT('JoinClosestTrack : ', TO_STRING(TrackToJoin));
			LogEntry.Accel	 := _MoveDynamics.A;
			LogEntry.Decel	 := _MoveDynamics.D;
			LogEntry.Jerk	 := _MoveDynamics.J;
			LogEntry.Vlocity := _MoveDynamics.V;
			UpdateLog();
			TaskState := TaskState + 10;
		ELSE
			TaskState := 99;
		END_IF
		
	50: //Watch feedback
		IF _PlanarFb.Done THEN
			TaskState := 60;
		ELSIF _PlanarFb.Error THEN
			_Error				:= TRUE;
			_ErrorID			:= _PlanarFb.ErrorId;
			_BlockingObjectInfo := _PlanarFb.objectInfo;
			TaskState			:= 0;
		END_IF

	60: //Task Complete
		THIS^._Done := TRUE;
		TaskState	:= 0;
		
	99:
		_Error := TRUE;
		_ErrorID := 9999;
		MoverStr := CONCAT('Mover ', TO_STRING(ipMover.MoverIndex));
		LogEntry.Command := CONCAT(CONCAT(MoverStr, ' : %s'), 'Join Closest Track - No Track Found');
		UpdateLog();
		TaskState	:= 0;
END_CASE


IF ExecuteWatchdog <> WatchdogCheck THEN
	WatchdogCheck := ExecuteWatchdog;
ELSE
	HasRun			:= FALSE;
	ExecuteWatchdog := 0;
END_IF
END_METHOD

END_FUNCTION_BLOCK

// Mover/TaskClasses/FB_JoinTrack
FUNCTION_BLOCK FB_JoinTrack EXTENDS FB_MoverTaskResult
VAR
	JoinTrackOptions : ST_JoinTrackOptions;
END_VAR

METHOD Execute : I_PlanarTaskResult
VAR_INPUT
	ipTrack		   : I_XPlanarTrack;
	UseOrientation : BOOL;
	MoveDynamics   : REFERENCE TO DynamicConstraint_PathXYZ;
END_VAR
IF NOT HasRun AND (ipMover.Status.CommandMode <> MC_Planar_Mover_Command_Mode.OnTrack) THEN
	_Done	 := FALSE;
	_Error	 := FALSE;
	_Busy	 := FALSE;
	_ErrorID := 0;
	JoinTrackOptions.useOrientation := UseOrientation;
	ipMover.pm.JoinTrack(_PlanarFb,
					ipTrack.pm,
					MoveDynamics,
					JoinTrackOptions);

	//Update mover command log				
	LogEntry.Command := CONCAT('JoinTrack : ', TO_STRING(ipTrack.Index));
	LogEntry.Accel	 := MoveDynamics.A;
	LogEntry.Decel	 := MoveDynamics.D;
	LogEntry.Jerk	 := MoveDynamics.J;
	LogEntry.Vlocity := MoveDynamics.V;
	UpdateLog();
	HasRun := TRUE;
END_IF

Execute := THIS^;

//Heartbeat that the method is active
ExecuteWatchdog := ExecuteWatchdog + 1;
END_METHOD

END_FUNCTION_BLOCK

// Mover/TaskClasses/FB_LeaveMovementArea
FUNCTION_BLOCK FB_LeaveMovementArea EXTENDS FB_MoverTaskResult
VAR
	MovementAreaParameters : EnterOrLeaveMovementAreaParameters;
	LeaveMvmtArea		   : BOOL;
END_VAR

METHOD Execute : I_PlanarTaskResult
IF NOT HasRun THEN
	_Done								   := FALSE;
	_Error								   := FALSE;
	_Busy								   := FALSE;
	_ErrorID							   := 0;
	MovementAreaParameters.MovementAreaOID := 0;
	LeaveMvmtArea						   := TRUE;
	HasRun								   := TRUE;

	//Update mover command log				
	LogEntry.Command := 'Remove From Movement Area';
	UpdateLog();
END_IF

Execute := THIS^;

//Heartbeat that the method is active
ExecuteWatchdog := ExecuteWatchdog + 1;
END_METHOD

METHOD Update
VAR_INST
	WatchdogCheck : UDINT;
END_VAR
//State logic for the task
CASE TaskState OF
	0: // Init
		_Busy := FALSE;
		IF LeaveMvmtArea THEN
			_Done		  := FALSE;
			_Error		  := FALSE;
			_ErrorID	  := 0;
			_Busy		  := TRUE;
			LeaveMvmtArea := FALSE;
			TaskState	  := TaskState + 10;
		END_IF

	10:  //Remove Mover from Movement Area
		IF ipMover.Utility.SetMovementArea(MovementAreaParameters) THEN
			TaskState := TaskState + 10;
		END_IF

	20:
		IF SUCCEEDED(MovementAreaParameters.Result) THEN
			_Done	  := TRUE;
			TaskState := 0;
		ELSIF FAILED(MovementAreaParameters.Result) THEN
			_Error	  := TRUE;
			_ErrorID  := TO_UDINT(MovementAreaParameters.Result);
			TaskState := 0;
		END_IF
END_CASE

RT_ADSWarn(CLK := _Error);
IF RT_ADSWarn.Q THEN
	ADSLOGSTR(ADSLOG_MSGTYPE_WARN, CONCAT('Mover ', ipMover.MoverBTN), CONCAT(_TaskName, CONCAT('Error ', TO_STRING(_ErrorId))));
END_IF

IF ExecuteWatchdog <> WatchdogCheck THEN
	WatchdogCheck := ExecuteWatchdog;
ELSE
	HasRun			:= FALSE;
	ExecuteWatchdog := 0;
END_IF
END_METHOD

END_FUNCTION_BLOCK

// Mover/TaskClasses/FB_LeaveTrack
{attribute 'no_assign_warning'}
FUNCTION_BLOCK FB_LeaveTrack EXTENDS FB_MoverTaskResult
VAR
	LeaveTrackOptions : ST_LeaveTrackOptions;
END_VAR

METHOD Execute : I_PlanarTaskResult
VAR_INPUT
	TargetPositionX : LREAL;
	TargetPositionY : LREAL;
	UseOrientation	: BOOL;
	MoveDynamics	: REFERENCE TO DynamicConstraint_PathXYZ;
END_VAR

VAR_INST
	Target : PositionXYC;
END_VAR
IF NOT HasRun AND ipMover.Status.CommandMode = MC_Planar_Mover_Command_Mode.OnTrack THEN
	_Done							 := FALSE;
	_Error							 := FALSE;
	_Busy							 := FALSE;
	_ErrorID						 := 0;
	LeaveTrackOptions.useOrientation := UseOrientation;
	Target.SetValuesXYC(TargetPositionX, TargetPositionY, ActualPosition.c);
	ipMover.pm.LeaveTrack(_PlanarFb,
						  Target,
						  MoveDynamics,
						  LeaveTrackOptions);

	//Update mover command log				
	LogEntry.Command := CONCAT('LeaveTrackTo : ', CONCAT(CONCAT('X= ', TO_STRING(TargetPositionX)), CONCAT(' Y= ', TO_STRING(TargetPositionY))));
	LogEntry.Accel	 := MoveDynamics.A;
	LogEntry.Decel	 := MoveDynamics.D;
	LogEntry.Jerk	 := MoveDynamics.J;
	LogEntry.Vlocity := MoveDynamics.V;
	UpdateLog();
	HasRun := TRUE;
END_IF

Execute := THIS^;

//Heartbeat that the method is active
ExecuteWatchdog := ExecuteWatchdog + 1;
END_METHOD

END_FUNCTION_BLOCK

// Mover/TaskClasses/FB_MoveA
FUNCTION_BLOCK FB_MoveA EXTENDS FB_MoverTaskResult
VAR
	PositionBuffer	: LREAL;
END_VAR

METHOD Execute : I_PlanarTaskResult
VAR_INPUT
	Position	 : LREAL;
	MoveDynamics : REFERENCE TO DynamicConstraint_Coordinates;
END_VAR
IF NOT HasRun OR (Position <> PositionBuffer) THEN
	_Done	 := FALSE;
	_Error	 := FALSE;
	_Busy	 := FALSE;
	_ErrorID := 0;
	ipMover.pm.MoveA(_PlanarFb, Position, MoveDynamics);

	//Update mover command log				
	LogEntry.Command := CONCAT('MoveA : ', TO_STRING(Position));
	LogEntry.Accel	 := MoveDynamics.GetA(Coord_Mcs_A1);
	LogEntry.Decel	 := MoveDynamics.GetD(Coord_Mcs_A1);
	LogEntry.Jerk	 := MoveDynamics.GetJ(Coord_Mcs_A1);
	LogEntry.Vlocity := MoveDynamics.GetV(Coord_Mcs_A1);
	UpdateLog();
	
	//Update call buffers
	PositionBuffer := Position;
	HasRun := TRUE;
END_IF

Execute := THIS^;

//Heartbeat that the method is active
ExecuteWatchdog := ExecuteWatchdog + 1;
END_METHOD

END_FUNCTION_BLOCK

// Mover/TaskClasses/FB_MoveB
FUNCTION_BLOCK FB_MoveB EXTENDS FB_MoverTaskResult
VAR
	PositionBuffer	: LREAL;
END_VAR

METHOD Execute : I_PlanarTaskResult
VAR_INPUT
	Position	 : LREAL;
	MoveDynamics : REFERENCE TO DynamicConstraint_Coordinates;
END_VAR
IF NOT HasRun OR (Position <> PositionBuffer) THEN
	_Done	 := FALSE;
	_Error	 := FALSE;
	_Busy	 := FALSE;
	_ErrorID := 0;
	ipMover.pm.MoveB(_PlanarFb, Position, MoveDynamics);

	//Update mover command log				
	LogEntry.Command := CONCAT('MoveB : ', TO_STRING(Position));
	LogEntry.Accel	 := MoveDynamics.GetA(Coord_Mcs_B1);
	LogEntry.Decel	 := MoveDynamics.GetD(Coord_Mcs_B1);
	LogEntry.Jerk	 := MoveDynamics.GetJ(Coord_Mcs_B1);
	LogEntry.Vlocity := MoveDynamics.GetV(Coord_Mcs_B1);
	UpdateLog();
	
	//Update call buffers
	PositionBuffer := Position;
	HasRun := TRUE;
END_IF

Execute := THIS^;

//Heartbeat that the method is active
ExecuteWatchdog := ExecuteWatchdog + 1;
END_METHOD

END_FUNCTION_BLOCK

// Mover/TaskClasses/FB_MoveToPosition
{attribute 'no_assign_warning'}
FUNCTION_BLOCK FB_MoveToPosition EXTENDS FB_MoverTaskResult
VAR
	MoveOptions		: ST_MoveToPositionOptions;
	MoverPosition	: MoverVector;
	Position		: PositionXYC;
	XPositionBuffer : LREAL;
	YPositionBuffer : LREAL;
END_VAR

METHOD Execute : I_PlanarTaskResult
VAR_INPUT
	XPosition	 : LREAL;
	YPosition	 : LREAL;
	MoveDynamics : REFERENCE TO DynamicConstraint_PathXYZ;
END_VAR
IF NOT HasRun OR ((XPosition <> XPositionBuffer) OR (YPosition <> YPositionBuffer)) THEN
	_Done		  := FALSE;
	_Error		  := FALSE;
	_Busy		  := FALSE;
	_ErrorID	  := 0;
	MoverPosition := ipMover.pm.MCTOPLC.SET.SetPos;
	Position.SetValuesXYC(XPosition, YPosition, MoverPosition.c);
	ipMover.pm.MoveToPosition(_PlanarFb,
							  Position,
							  MoveDynamics,
							  MoveOptions);

	//Update mover command log				
	LogEntry.Command := CONCAT('MoveToPosition : ', CONCAT(CONCAT('X= ', TO_STRING(XPosition)), CONCAT(' Y= ', TO_STRING(YPosition))));
	LogEntry.Accel	 := MoveDynamics.A;
	LogEntry.Decel	 := MoveDynamics.D;
	LogEntry.Jerk	 := MoveDynamics.J;
	LogEntry.Vlocity := MoveDynamics.V;
	UpdateLog();

	//Update call buffers
	XPositionBuffer := XPosition;
	YPositionBuffer := YPosition;
	HasRun			:= TRUE;
END_IF

Execute := THIS^;

//Heartbeat that the method is active
ExecuteWatchdog := ExecuteWatchdog + 1;
END_METHOD

END_FUNCTION_BLOCK

// Mover/TaskClasses/FB_MoveZ
FUNCTION_BLOCK FB_MoveZ EXTENDS FB_MoverTaskResult
VAR
	PositionBuffer	: LREAL;
END_VAR

METHOD Execute : I_PlanarTaskResult
VAR_INPUT
	Position	 : LREAL;
	MoveDynamics : REFERENCE TO DynamicConstraint_PathXYZ;
END_VAR
IF NOT HasRun OR (Position <> PositionBuffer) THEN
	_Done	 := FALSE;
	_Error	 := FALSE;
	_Busy	 := FALSE;
	_ErrorID := 0;
	ipMover.pm.MoveZ(_PlanarFb, Position, MoveDynamics);

	//Update mover command log				
	LogEntry.Command := CONCAT('MoveZ : ', TO_STRING(Position));
	LogEntry.Accel	 := MoveDynamics.A;
	LogEntry.Decel	 := MoveDynamics.D;
	LogEntry.Jerk	 := MoveDynamics.J;
	LogEntry.Vlocity := MoveDynamics.V;
	UpdateLog();
	
	//Update call buffers
	PositionBuffer := Position;
	HasRun := TRUE;
END_IF

Execute := THIS^;

//Heartbeat that the method is active
ExecuteWatchdog := ExecuteWatchdog + 1;
END_METHOD

END_FUNCTION_BLOCK

// Mover/TaskClasses/FB_ResetMover
FUNCTION_BLOCK FB_ResetMover EXTENDS FB_MoverTaskResult
VAR
END_VAR

METHOD Execute : I_PlanarTaskResult
IF NOT HasRun THEN
	_Done		:= FALSE;
	_Error		:= FALSE;
	_Busy		:= FALSE;
	_ErrorID	:= 0;
	ipMover.pm.Reset(_PlanarFb);
	HasRun := TRUE;
END_IF

Execute := THIS^;

//Heartbeat that the method is active
ExecuteWatchdog := ExecuteWatchdog + 1;
END_METHOD

END_FUNCTION_BLOCK

// Mover/TaskClasses/FB_Rotate
FUNCTION_BLOCK FB_Rotate EXTENDS FB_MoverTaskResult
VAR
	RotateOptions : ST_MoveCOptions;
	PositionBuffer	: LREAL;
	TurnsBuffer		: DINT;
END_VAR

METHOD Execute : I_PlanarTaskResult
VAR_INPUT
	Distance	   : LREAL;
	NumberOfTurns  : DINT;
	Direction	   : Tc3_Mc3PlanarMotion.MC_DIRECTION;
	RotateDynamics : REFERENCE TO DynamicConstraint_Coordinates;
END_VAR
IF NOT HasRun OR ((Distance <> PositionBuffer) OR (NumberOfTurns <> TurnsBuffer)) THEN
	_Done						  := FALSE;
	_Error						  := FALSE;
	_Busy						  := FALSE;
	_ErrorID					  := 0;
	RotateOptions.direction		  := Direction;
	RotateOptions.additionalTurns := TO_UDINT(NumberOfTurns);
	ipMover.pm.MoveC(_PlanarFb,
					 Distance,
					 RotateDynamics,
					 RotateOptions);

	//Update mover command log				
	LogEntry.Command := CONCAT('MoveC : ', CONCAT(TO_STRING(Distance), CONCAT(' : Turns ', TO_STRING(NumberOfTurns))));
	LogEntry.Accel	 := RotateDynamics.GetA(Coord_Mcs_C1);
	LogEntry.Decel	 := RotateDynamics.GetD(Coord_Mcs_C1);
	LogEntry.Jerk	 := RotateDynamics.GetJ(Coord_Mcs_C1);
	LogEntry.Vlocity := RotateDynamics.GetV(Coord_Mcs_C1);
	UpdateLog();

	//Update call buffers
	PositionBuffer := Distance;
	TurnsBuffer	   := NumberOfTurns;
	HasRun		   := TRUE;
END_IF

Execute := THIS^;

//Heartbeat that the method is active
ExecuteWatchdog := ExecuteWatchdog + 1;
END_METHOD

END_FUNCTION_BLOCK

// Mover/TaskClasses/FB_RunExternalSetpointAbsoluteMode
FUNCTION_BLOCK FB_RunExternalSetpointAbsoluteMode EXTENDS FB_MoverTaskResult
VAR
	ExternalSetpointGenerationOptions : ST_ExternalSetpointGenerationOptions;
END_VAR

METHOD Execute : I_PlanarTaskResult
VAR_INPUT
	Position	 : MoverVector;
	Velocity	 : MoverVector;
	Acceleration : MoverVector;
END_VAR
IF NOT HasRun THEN
	_Done								   := FALSE;
	_Error								   := FALSE;
	_Busy								   := FALSE;
	_ErrorID							   := 0;
	ExternalSetpointGenerationOptions.mode := MC_EXTERNAL_SET_POSITION_MODE.Absolute;
	ipMover.pm.StartExternalSetpointGeneration(_PlanarFb, ExternalSetpointGenerationOptions);

	//Update mover command log				
	LogEntry.Command := CONCAT('Follow External setpoint started at : ', CONCAT(CONCAT('X= ', TO_STRING(Position.x)), CONCAT(' Y= ', TO_STRING(Position.y))));
	UpdateLog();
	HasRun := TRUE;
END_IF

ipMover.pm.SetExternalSetpoint(Position, Velocity, Acceleration);
Execute := THIS^;

//Heartbeat that the method is active
ExecuteWatchdog := ExecuteWatchdog + 1;
END_METHOD

END_FUNCTION_BLOCK

// Mover/TaskClasses/FB_RunExternalSetpointRelativeMode
FUNCTION_BLOCK FB_RunExternalSetpointRelativeMode EXTENDS FB_MoverTaskResult
VAR
	ExternalSetpointGenerationOptions : ST_ExternalSetpointGenerationOptions;
END_VAR

METHOD Execute : I_PlanarTaskResult
VAR_INPUT
	Position	 : MoverVector;
	Velocity	 : MoverVector;
	Acceleration : MoverVector;
END_VAR
IF NOT HasRun THEN
	_Done								   := FALSE;
	_Error								   := FALSE;
	_Busy								   := FALSE;
	_ErrorID							   := 0;
	ExternalSetpointGenerationOptions.mode := MC_EXTERNAL_SET_POSITION_MODE.Relative;
	ipMover.pm.StartExternalSetpointGeneration(_PlanarFb, ExternalSetpointGenerationOptions);

	//Update mover command log				
	LogEntry.Command := CONCAT('Follow External setpoint started at : ', CONCAT(CONCAT('X= ', TO_STRING(Position.x)), CONCAT(' Y= ', TO_STRING(Position.y))));
	UpdateLog();
	HasRun := TRUE;
END_IF

ipMover.pm.SetExternalSetpoint(Position, Velocity, Acceleration);
Execute := THIS^;

//Heartbeat that the method is active
ExecuteWatchdog := ExecuteWatchdog + 1;
END_METHOD

END_FUNCTION_BLOCK

// Mover/TaskClasses/FB_SquareUp
{attribute 'no_assign_warning'} 
FUNCTION_BLOCK FB_SquareUp EXTENDS FB_MoverTaskResult
VAR
	RotateOptions	: Tc3_Mc3PlanarMotion.ST_MoveCOptions;
	_RotateDynamics : REFERENCE TO Tc3_Physics.DynamicConstraint_Coordinates;
	_MoveDynamics	: REFERENCE TO Tc3_Physics.DynamicConstraint_PathXYZ;
	_Distance		: LREAL;
	SquareUp		: BOOL;
END_VAR

METHOD Execute : I_PlanarTaskResult
VAR_INPUT
	Distance	   : LREAL;
	RotateDynamics : REFERENCE TO Tc3_Physics.DynamicConstraint_Coordinates;
	MoveDynamics   : REFERENCE TO Tc3_Physics.DynamicConstraint_PathXYZ;
END_VAR
IF NOT HasRun THEN
	_Done			:= FALSE;
	_Error			:= FALSE;
	_Busy			:= FALSE;
	_ErrorID		:= 0;
	_Distance		:= Distance;
	_RotateDynamics REF= RotateDynamics;
	_MoveDynamics	ref= MoveDynamics;
	SquareUp		:= TRUE;
	HasRun			:= TRUE;
END_IF

Execute := THIS^;

//Heartbeat that the method is active
ExecuteWatchdog := ExecuteWatchdog + 1;
END_METHOD

METHOD Update
VAR_INST
	WatchdogCheck : UDINT;
END_VAR
//***Overwriting the update method because this task contains a state machine that must be monitored cyclically.***
_PlanarFb.Update();

//State logic for the task
CASE TaskState OF
	0: // Init
		_Busy := FALSE;
		IF SquareUp THEN
			_Done	  := FALSE;
			_Error	  := FALSE;
			_Aborted  := FALSE;
			_ErrorID  := 0;
			_Busy	  := TRUE;
			SquareUp  := FALSE;
			TaskState := TaskState + 10;
		END_IF

	10: //Rotate C to closest quarter angle
		RotateOptions.direction		  := Tc3_Mc3PlanarMotion.MC_DIRECTION.mcDirectionShortestWay;
		RotateOptions.additionalTurns := 0;
		ipMover.pm.MoveC(_PlanarFb,
						 _Distance,
						 _RotateDynamics,
						 RotateOptions);

		//Update mover command log				
		LogEntry.Command := CONCAT('MoveC : ', TO_STRING(_Distance));
		LogEntry.Accel	 := _RotateDynamics.GetA(Coord_Mcs_C1);
		LogEntry.Decel	 := _RotateDynamics.GetD(Coord_Mcs_C1);
		LogEntry.Jerk	 := _RotateDynamics.GetJ(Coord_Mcs_C1);
		LogEntry.Vlocity := _RotateDynamics.GetV(Coord_Mcs_C1);
		UpdateLog();
		TaskState := TaskState + 10;

	20: //Watch rotate feedback
		IF _PlanarFb.Done THEN
			TaskState := TaskState + 10;
		ELSIF _PlanarFb.Error THEN
			TaskState := 999;
		ELSIF _PlanarFb.Aborted THEN
			_Aborted  := TRUE;
			TaskState := 0;
		END_IF

	30: //Move A Axis to 0
		ipMover.pm.MoveA(_PlanarFb, 0.0, _MoveDynamics);

		//Update mover command log				
		LogEntry.Command := CONCAT('Move A : ', TO_STRING(0.0));
		LogEntry.Accel	 := _MoveDynamics.A;
		LogEntry.Decel	 := _MoveDynamics.D;
		LogEntry.Jerk	 := _MoveDynamics.J;
		LogEntry.Vlocity := _MoveDynamics.V;
		UpdateLog();
		TaskState := TaskState + 10;

	40: //A Axis move feedback
		IF _PlanarFb.Done THEN
			TaskState := TaskState + 10;
		ELSIF _PlanarFb.Error THEN
			TaskState := 999;
		ELSIF _PlanarFb.Aborted THEN
			_Aborted := TRUE;
			TaskState := 0;
		END_IF

	50: //Move B Axis to 0
		ipMover.pm.MoveB(_PlanarFb, 0.0, _MoveDynamics);

		//Update mover command log				
		LogEntry.Command := CONCAT('Move B : ', TO_STRING(0.0));
		LogEntry.Accel	 := _MoveDynamics.A;
		LogEntry.Decel	 := _MoveDynamics.D;
		LogEntry.Jerk	 := _MoveDynamics.J;
		LogEntry.Vlocity := _MoveDynamics.V;
		UpdateLog();
		TaskState := TaskState + 10;

	60: //A Axis move feedback
		IF _PlanarFb.Done THEN
			TaskState := TaskState + 10;
		ELSIF _PlanarFb.Error THEN
			TaskState := 999;
		ELSIF _PlanarFb.Aborted THEN
			_Aborted := TRUE;
			TaskState := 0;
		END_IF

	70: //Task Complete
		_Done	  := TRUE;
		TaskState := 0;

	999: //Task Error
		_Error				:= TRUE;
		_ErrorID			:= _PlanarFb.ErrorId;
		_BlockingObjectInfo := _PlanarFb.objectInfo;
		TaskState			:= 0;
END_CASE

IF TaskState > 0 AND ipMover.Error THEN
	TaskState := 999;
END_IF

IF ExecuteWatchdog <> WatchdogCheck THEN
	WatchdogCheck := ExecuteWatchdog;
ELSE
	HasRun			:= FALSE;
	ExecuteWatchdog := 0;
END_IF
END_METHOD

END_FUNCTION_BLOCK

// Mover/TaskClasses/FB_StopExternalSetpoint
FUNCTION_BLOCK FB_StopExternalSetpoint EXTENDS FB_MoverTaskResult
VAR
	ExternalSetpointGenerationOptions : ST_ExternalSetpointGenerationOptions;
END_VAR

METHOD Execute : I_PlanarTaskResult
IF NOT HasRun THEN
	_Done	 := FALSE;
	_Error	 := FALSE;
	_Busy	 := FALSE;
	_ErrorID := 0;
	ipMover.pm.StopExternalSetpointGeneration(_PlanarFb);

	//Update mover command log				
	LogEntry.Command := 'Stop external setpoint';
	UpdateLog();
	HasRun := TRUE;
END_IF

Execute := THIS^;

//Heartbeat that the method is active
ExecuteWatchdog := ExecuteWatchdog + 1;
END_METHOD

END_FUNCTION_BLOCK

// Mover/TaskClasses/FB_TrackMove
{attribute 'no_assign_warning'} 
FUNCTION_BLOCK FB_TrackMove EXTENDS FB_MoverTaskResult
VAR
	DynMove			   : DynamicConstraint_PathXY;
	MoveOnTrackOptions : ST_MoveOnTrackOptions;
	MoverSetPos		   : MoverVector;
	OnTrackPos		   : LREAL;
END_VAR

METHOD Execute : I_PlanarTaskResult
VAR_INPUT
	Position	 : LREAL;
	Gap			 : LREAL;
	TrackSegment : I_XPlanarTrack;
	MoveDynamics : REFERENCE TO DynamicConstraint_PathXY;
	Direction	 : Tc3_Mc3PlanarMotion.MC_DIRECTION;
END_VAR
IF NOT HasRun AND (ipMover.Status.CommandMode = MC_Planar_Mover_Command_Mode.OnTrack OR ipMover.Status.CommandMode = MC_Planar_Mover_Command_Mode.CRotationOnTrack) THEN
	_Done		:= FALSE;
	_Error		:= FALSE;
	_Busy		:= FALSE;
	_ErrorID	:= 0;
	MoveOnTrackOptions.gap		 := Gap;
	MoveOnTrackOptions.direction := Direction;
	ipMover.pm.MoveOnTrack(_PlanarFb,
					  TrackSegment.pm,
					  Position,
					  MoveDynamics,
					  MoveOnTrackOptions);

	//Update mover command log				
	LogEntry.Command := CONCAT('MoveOnTrack : ', CONCAT(CONCAT('ID : ', TO_STRING(TrackSegment.Index)), CONCAT(' Pos ', TO_STRING(Position))));
	LogEntry.Accel	 := MoveDynamics.A;
	LogEntry.Decel	 := MoveDynamics.D;
	LogEntry.Jerk	 := MoveDynamics.J;
	LogEntry.Vlocity := MoveDynamics.V;
	UpdateLog();
	HasRun := TRUE;
END_IF

Execute := THIS^;

//Heartbeat that the method is active
ExecuteWatchdog := ExecuteWatchdog + 1;
END_METHOD

END_FUNCTION_BLOCK

// Mover/TaskClasses/FB_TrackMoveXY
{attribute 'no_assign_warning'}
FUNCTION_BLOCK FB_TrackMoveXY EXTENDS FB_MoverTaskResult
VAR
	DynMove			   : DynamicConstraint_PathXY;
	MoveOnTrackOptions : ST_MoveOnTrackOptions;
END_VAR

METHOD Execute : I_PlanarTaskResult
VAR_INPUT
	PositionX	 : LREAL;
	PositionY	 : LREAL;
	Gap			 : LREAL;
	TrackSegment : I_XPlanarTrack;
	MoveDynamics : REFERENCE TO DynamicConstraint_PathXY;
	Direction	 : Tc3_Mc3PlanarMotion.MC_DIRECTION;
END_VAR

VAR_INST
	Position		: PositionXYC;
	SetPosition		: MoverVector;
	OnTrackPosition : LREAL;
END_VAR
IF NOT HasRun AND (ipMover.Status.CommandMode = MC_Planar_Mover_Command_Mode.OnTrack OR ipMover.Status.CommandMode = MC_Planar_Mover_Command_Mode.CRotationOnTrack) THEN
	_Done		:= FALSE;
	_Error		:= FALSE;
	_Busy		:= FALSE;
	_ErrorID	:= 0;
	SetPosition := ipMover.pm.MCTOPLC.SET.SetPos;
	Position.SetValuesXY(PositionX, PositionY);
	MoveOnTrackOptions.gap		 := Gap;
	MoveOnTrackOptions.direction := Direction;
	OnTrackPosition				 := TrackSegment.GetTrackPositionAt(Position);
	ipMover.pm.MoveOnTrack(_PlanarFb,
					  TrackSegment.pm,
					  OnTrackPosition,
					  MoveDynamics,
					  MoveOnTrackOptions);

	//Update mover command log				
	LogEntry.Command := CONCAT('MoveOnTrack : ', CONCAT(CONCAT('ID : ', TO_STRING(TrackSegment.Index)), CONCAT(' Pos ', TO_STRING(OnTrackPosition))));
	LogEntry.Accel	 := MoveDynamics.A;
	LogEntry.Decel	 := MoveDynamics.D;
	LogEntry.Jerk	 := MoveDynamics.J;
	LogEntry.Vlocity := MoveDynamics.V;
	UpdateLog();
	HasRun := TRUE;
END_IF

Execute := THIS^;

//Heartbeat that the method is active
ExecuteWatchdog := ExecuteWatchdog + 1;
END_METHOD

END_FUNCTION_BLOCK

// Mover/FB_XPlanarMover
{attribute 'no_assign'}
{attribute 'no_explicit_call' := 'do not call this POU directly'}
FUNCTION_BLOCK FB_XPlanarMover EXTENDS FB_CyclicFB IMPLEMENTS I_XPlanarMover, I_MoveCommands, I_MoveDynamics
VAR
	_Mover		: Tc3_MC3PlanarMotion.MC_PlanarMover;
	_ObjectInfo : Tc3_Mc3PlanarMotion.PlanarObjectInfo;
	_std		: CDT_MCTOPLC_PLANAR_MOVER_STD;

	//Command Log
	_CommandLog : ARRAY[0..SystemParameters.MAX_LOG_COUNT] OF ST_CommandLog;

	//Mover Task Declarations
	EnableMover						: FB_Enable							 := (Mover := THIS^, TaskName := 'Enable');
	DisableMover					: FB_Disable						 := (Mover := THIS^, TaskName := 'Disable');
	HaltMover						: FB_Halt							 := (Mover := THIS^, TaskName := 'Halt');
	JoinMoverToTrack				: FB_JoinTrack						 := (Mover := THIS^, TaskName := 'JoinTrack');
	JoinToClosestTrack				: FB_JoinClosestTrack				 := (Mover := THIS^, TaskName := 'JoinClosestTrack');
	LeaveMoverFromTrack				: FB_LeaveTrack						 := (Mover := THIS^, TaskName := 'LeaveTrack');
	ResetMover						: FB_ResetMover						 := (Mover := THIS^, TaskName := 'Reset');
	MoveOnTrackXY					: FB_TrackMoveXY					 := (Mover := THIS^, TaskName := 'MoveOnTrack');
	MoveOnTrack						: FB_TrackMove						 := (Mover := THIS^, TaskName := 'MoveOnTrack');
	RotateMover						: FB_Rotate							 := (Mover := THIS^, TaskName := 'Rotate');
	ZMove							: FB_MoveZ							 := (Mover := THIS^, TaskName := 'MoveZ');
	AMove							: FB_MoveA							 := (Mover := THIS^, TaskName := 'MoveA');
	BMove							: FB_MoveB							 := (Mover := THIS^, TaskName := 'MoveB');
	MoveToPosition					: FB_MoveToPosition					 := (Mover := THIS^, TaskName := 'MoveToPosition');
	AddMoverToGroup					: FB_AddToGroup						 := (Mover := THIS^, TaskName := 'AddToGroup');
	SquareMover						: FB_SquareUp						 := (Mover := THIS^, TaskName := 'SquareUp');
	RunExternalSetpointRelativeMode : FB_RunExternalSetpointRelativeMode := (Mover := THIS^, TaskName := 'Run external setpoint relative mode');
	RunExternalSetpointAbsoluteMode : FB_RunExternalSetpointAbsoluteMode := (Mover := THIS^, TaskName := 'Run external setpoint absolute mode');
	StopExternalSetpoint			: FB_StopExternalSetpoint			 := (Mover := THIS^, TaskName := 'Stop external setpoint');
	EnterMvmtAreaTask				: FB_EnterMovementArea				 := (Mover := THIS^, TaskName := 'EnterMovementArea');
	LeaveMvmtAreaTask				: FB_LeaveMovementArea				 := (Mover := THIS^, TaskName := 'LeaveMovementArea');
	InvalidCommandResult			: FB_ResultBase						 := (Busy := FALSE, Error := TRUE, ErrorID := 9999);

	//Internal Vars
	_MoveDynamics		 : ST_MoveDynamics;
	_RotateDynamics		 : ST_MoveDynamics;
	_TiltDynamics		 : ST_MoveDynamics;
	_DynMove			 : Tc3_Physics.DynamicConstraint_PathXYZ;
	_DynRotate			 : Tc3_Physics.DynamicConstraint_Coordinates;
	_DynTrackMove		 : Tc3_Physics.DynamicConstraint_PathXY;
	_DynHalt			 : Tc3_Physics.DynamicConstraint_Coordinates;
	_Gap				 : LREAL;
	_MoverIndex			 : UDINT;
	_TrackId			 : UDINT;
	_MoverBTN			 : STRING;
	_IdentifiedBTN		 : STRING;
	_MoverType			 : XPlanarMoverType;
	_InStation			 : BOOL;
	ipDestination		 : I_XPlanarStation;
	ipMoverTcIo			 : I_TcIoXPlanarMover;
	_ModuloPosC			 : LREAL;
	TypeIsRead			 : BOOL;
	ClosestSquarePos	 : LREAL;
	_MoverActPos		 : MoverVector;
	_ClosestQuarterAngle : LREAL;
	_AtRotationPosition	 : BOOL;
	UpdateMoveDynamics	 : BOOL;
	UpdateRotateDynamics : BOOL;
	UpdateTiltDynamics	 : BOOL;
END_VAR

{attribute 'TcRpcEnable'}
METHOD FreeMove : I_PlanarTaskResult
VAR_INPUT
	XPosition : LREAL;
	YPosition : LREAL;
END_VAR

VAR_INST
	Position : PositionXYC;
END_VAR
FreeMove := MoveToPosition.Execute(XPosition, YPosition, _DynMove);
END_METHOD

{attribute 'TcRpcEnable'}
METHOD JoinClosestTrack : I_PlanarTaskResult
VAR_INPUT
	UseOrientation : BOOL;
END_VAR
JoinClosestTrack := JoinToClosestTrack.Execute(UseOrientation, _DynMove);
END_METHOD

{attribute 'TcRpcEnable'}
METHOD JoinTrack : I_PlanarTaskResult
VAR_INPUT
	ipTrack		   : I_XPlanarTrack;
	UseOrientation : BOOL;
END_VAR
JoinTrack := JoinMoverToTrack.Execute(ipTrack, UseOrientation, _DynMove);
END_METHOD

{attribute 'TcRpcEnable'}
METHOD LeaveTrack : I_PlanarTaskResult
VAR_INPUT
	DestinationX   : LREAL;
	DestinationY   : LREAL;
	UseOrientation : BOOL;
END_VAR

VAR_INST
	Destination : PositionXYC;
END_VAR
LeaveTrack := LeaveMoverFromTrack.Execute(DestinationX,
										  DestinationY,
										  UseOrientation,
										  _DynMove);
END_METHOD

{attribute 'TcRpcEnable'}
METHOD Rotate : I_PlanarTaskResult
VAR_INPUT
	Position		: LREAL;
	AdditionalTurns : DINT;
END_VAR

VAR
	Direction : Tc3_Mc3PlanarMotion.MC_DIRECTION;
END_VAR
IF AdditionalTurns < 0 OR Position < 0 THEN
	Direction := Tc3_Mc3PlanarMotion.MC_DIRECTION.mcDirectionNegative;
ELSIF Position = 0 AND AdditionalTurns = 0 THEN
	Direction := Tc3_Mc3PlanarMotion.MC_DIRECTION.mcDirectionShortestWay;
ELSE
	Direction := Tc3_Mc3PlanarMotion.MC_DIRECTION.mcDirectionPositive;
END_IF

IF _AtRotationPosition OR ((Position >= -10 OR Position <= 10) AND AdditionalTurns = 0) THEN
	Rotate := RotateMover.Execute(ABS(Position),
								  ABS(AdditionalTurns),
								  Direction,
								  _DynRotate);
ELSE
	Rotate := InvalidCommandResult;
END_IF
END_METHOD

{attribute 'TcRpcEnable'}
METHOD RunExternalSpAbsoluteMode : I_PlanarTaskResult
VAR_INPUT
	Position	 : MoverVector;
	Velocity	 : MoverVector;
	Acceleration : MoverVector;
END_VAR
RunExternalSpAbsoluteMode := RunExternalSetpointAbsoluteMode.Execute(Position,Velocity,Acceleration);
END_METHOD

{attribute 'TcRpcEnable'}
METHOD RunExternalSpRelativeMode : I_PlanarTaskResult
VAR_INPUT
	Position	 : MoverVector;
	Velocity	 : MoverVector;
	Acceleration : MoverVector;
END_VAR
RunExternalSpRelativeMode := RunExternalSetpointRelativeMode.Execute(Position,Velocity,Acceleration);
END_METHOD

{attribute 'TcRpcEnable'}
METHOD SendToStation : I_PlanarTaskResult
VAR_INPUT
	Destination : I_XPlanarStation;
END_VAR

VAR_INST
	CorrectedPos : PositionXYC;
	OnTrackPos	 : LREAL;
END_VAR
ipDestination := Destination; //Update the destination field of the mover
IF _Mover.MCTOPLC.STD.CommandMode = MC_PLANAR_MOVER_COMMAND_MODE.OnTrack THEN
	IF Destination.TrackID <> 0 THEN
		SendToStation := MoveOnTrackXY.Execute(Destination.Position.x,
											   Destination.Position.y,
											   _Gap,
											   ip.Tracks[Destination.TrackID],
											   _DynTrackMove,
											   Tc3_Mc3PlanarMotion.MC_DIRECTION.mcDirectionPositive);

		IF SystemParameters.EnableCommandTracing THEN
			THIS^.Trace(CONCAT(CONCAT('Mover ', TO_STRING(_MoverIndex)), CONCAT(', ', CONCAT('TrackMoveToStation ', TO_STRING(Destination.ID)))));
		END_IF
	ELSE
		SendToStation := InvalidCommandResult;
	END_IF
ELSIF _Mover.MCTOPLC.STD.CommandMode = MC_PLANAR_MOVER_COMMAND_MODE.FreeMovement THEN
	CorrectedPos.SetValuesXYC(Destination.Position.x, Destination.Position.y, _MoverActPos.c);
	SendToStation := MoveToPosition.Execute(Destination.Position.x, Destination.Position.y, _DynMove);
	IF SystemParameters.EnableCommandTracing THEN
		THIS^.Trace(CONCAT(CONCAT('Mover ', TO_STRING(_MoverIndex)), CONCAT(', ', CONCAT('FreeMoveToStation ', TO_STRING(Destination.ID)))));
	END_IF
ELSE
	SendToStation := InvalidCommandResult;
END_IF
END_METHOD

{attribute 'TcRpcEnable'}
METHOD SquareUp : I_PlanarTaskResult
VAR_INST
	Result		 : FB_ResultBase;
END_VAR
SquareUp := SquareMover.Execute(_ClosestQuarterAngle, _DynRotate, _DynMove);
END_METHOD

{attribute 'TcRpcEnable'}
METHOD StopExternalSp : I_PlanarTaskResult
StopExternalSp := StopExternalSetpoint.Execute();
END_METHOD

METHOD TiltA : I_PlanarTaskResult
VAR_INPUT
	Position : LREAL;
END_VAR
TiltA := AMove.Execute(Position, _DynRotate);
END_METHOD

METHOD TiltB : I_PlanarTaskResult
VAR_INPUT
	Position : LREAL;
END_VAR
TiltB := BMove.Execute(Position, _DynRotate);
END_METHOD

{attribute 'TcRpcEnable'}
METHOD TrackMove : I_PlanarTaskResult
VAR_INPUT
	Position : LREAL;
	Gap		  : LREAL;
	Track	  : I_XPlanarTrack;
	Direction : Tc3_Mc3PlanarMotion.MC_DIRECTION;
END_VAR

VAR
	WorkingGap : LREAL;
END_VAR
IF Gap > 0 THEN
	WorkingGap := Gap;
ELSE
	WorkingGap := _Gap;
END_IF

IF Track <> 0 THEN
	TrackMove := MoveOnTrack.Execute(Position,
									 WorkingGap,
									 Track,
									 _DynTrackMove,
									 Direction);
ELSE
	TrackMove := InvalidCommandResult;
END_IF
END_METHOD

{attribute 'TcRpcEnable'}
METHOD TrackMoveXY : I_PlanarTaskResult
VAR_INPUT
	XPosition : LREAL;
	YPosition : LREAL;
	Gap		  : LREAL;
	Track	  : I_XPlanarTrack;
	Direction : Tc3_Mc3PlanarMotion.MC_DIRECTION;
END_VAR

VAR
	WorkingGap : LREAL;
END_VAR

VAR_INST
	Position   : PositionXYC;
	OnTrackPos : LREAL;
END_VAR
IF Gap > 0 THEN
	WorkingGap := Gap;
ELSE
	WorkingGap := _Gap;
END_IF

IF Track <> 0 THEN
	TrackMoveXY := MoveOnTrackXY.Execute(XPosition,
										 YPosition,
										 WorkingGap,
										 Track,
										 _DynTrackMove,
										 Direction);
ELSE
	TrackMoveXY := InvalidCommandResult;
END_IF
END_METHOD

{attribute 'TcRpcEnable'}
METHOD VerticalMove : I_PlanarTaskResult
VAR_INPUT
	Position : LREAL;
END_VAR
VerticalMove := ZMove.Execute(Position, _DynMove);
END_METHOD

{attribute 'suppress_wrn_C0410'}
PROPERTY Movement : REFERENCE TO ST_MoveDynamics
GET
Movement REF= _MoveDynamics;
UpdateMoveDynamics := TRUE;
END_GET
END_PROPERTY

{attribute 'suppress_wrn_C0410'}
PROPERTY Rotation : REFERENCE TO ST_MoveDynamics
GET
Rotation REF= _RotateDynamics;
UpdateRotateDynamics := true;
END_GET
END_PROPERTY

{attribute 'suppress_wrn_C0410'}
PROPERTY Tilt : REFERENCE TO ST_MoveDynamics
GET
Tilt REF= _TiltDynamics;
UpdateTiltDynamics := TRUE;
END_GET
END_PROPERTY

{attribute 'suppress_wrn_C0410'}
PROPERTY ActualPosition : REFERENCE TO MoverVector
GET
ActualPosition ref= _MoverActPos;
END_GET
END_PROPERTY

METHOD AddToGroup : I_PlanarTaskResult
VAR_INPUT
	PlanarGroup : REFERENCE TO MC_PlanarGroup;
END_VAR
AddToGroup := AddMoverToGroup.Execute(PlanarGroup);
END_METHOD

PROPERTY AtRotationPosition : BOOL
GET
AtRotationPosition := _AtRotationPosition;
END_GET
END_PROPERTY

{attribute 'suppress_wrn_C0410'}
PROPERTY CommandLog : REFERENCE TO ARRAY [0..SystemParameters.MAX_LOG_COUNT] of ST_CommandLog
GET
CommandLog ref= _CommandLog;
END_GET
END_PROPERTY

PROPERTY Destination : I_XPlanarStation
GET
Destination := ipDestination;
END_GET
SET
ipDestination := Destination;
END_SET
END_PROPERTY

{attribute 'TcRpcEnable'}
METHOD Disable : I_PlanarTaskResult
Disable := DisableMover.Execute();
END_METHOD

PROPERTY Dynamics : I_MoveDynamics
GET
Dynamics := THIS^;
END_GET
END_PROPERTY

{attribute 'TcRpcEnable'}
METHOD Enable : I_PlanarTaskResult
Enable := EnableMover.Execute();
END_METHOD

METHOD EnterMovementArea : I_PlanarTaskResult
VAR_INPUT
	PartId		: OTCID;
	PositionX	: LREAL;
	PositionY	: LREAL;
END_VAR
IF PartID = 0 AND PositionX < 0 OR PositionY < 0 THEN
	EnterMovementArea := InvalidCommandResult;
ELSE
	EnterMovementArea := EnterMvmtAreaTask.Execute(PartId, PositionX, PositionY);
END_IF
END_METHOD

PROPERTY Gap : LREAL
GET
Gap := _Gap;
END_GET
SET
_Gap := Gap;
END_SET
END_PROPERTY

METHOD Halt : I_PlanarTaskResult
Halt := HaltMover.Execute(_DynHalt);
END_METHOD

PROPERTY IdentifiedBTN : STRING
GET
IF ipMoverTcIo <> 0 THEN
	_IdentifiedBTN := ipMoverTcIo.GetIdentifiedMoverBtn();
END_IF

IdentifiedBTN := _IdentifiedBTN;
END_GET
SET
END_SET
END_PROPERTY

PROPERTY InStation : BOOL
GET
InStation := _InStation;
END_GET
SET
_InStation := InStation;
END_SET
END_PROPERTY

METHOD LeaveMovementArea : I_PlanarTaskResult
LeaveMovementArea := LeaveMvmtAreaTask.Execute();
END_METHOD

PROPERTY MoveCommand : I_MoveCommands
GET
MoveCommand := THIS^;
END_GET
END_PROPERTY

PROPERTY MoverBTN : STRING
GET
IF ipMoverTcIo <> 0 THEN
	_MoverBTN := ipMoverTcIo.GetBtn();
END_IF

MoverBTN := _MoverBTN;
END_GET
END_PROPERTY

PROPERTY MoverIndex : UDINT
GET
MoverIndex := _MoverIndex;
END_GET
SET
_MoverIndex := MoverIndex;
END_SET
END_PROPERTY

PROPERTY MoverType : XPlanarMoverType
GET
MoverType := _MoverType;
END_GET
SET
_MoverType := MoverType;
END_SET
END_PROPERTY

{attribute 'suppress_wrn_C0410'}
PROPERTY pm : REFERENCE TO MC_PlanarMover
GET
pm ref= _Mover;
END_GET
END_PROPERTY

//! @summary Clears error flags and error IDs for this component
{attribute 'TcRpcEnable'}
METHOD PUBLIC Reset : I_PlanarTaskResult
Reset := ResetMover.Execute();
END_METHOD

PROPERTY RotationModulo : LREAL
GET
RotationModulo := _ModuloPosC;
END_GET
END_PROPERTY

{attribute 'suppress_wrn_C0410'}
PROPERTY Status : REFERENCE TO CDT_MCTOPLC_PLANAR_MOVER_STD
GET
Status ref= _Std;
END_GET
END_PROPERTY

PROPERTY Utility : I_TcIoXPlanarMover
GET
IF ipMoverTcIo <> 0 THEN
	Utility := ipMoverTcIo;
END_IF
END_GET
SET
ipMoverTcIo := Utility;
END_SET
END_PROPERTY

//! @summary This method serves as the entry point for all underlying FB logic
METHOD PUBLIC CyclicLogic
//! @description This method should be called cyclically by descendant function blocks by invoking <c>SUPER^.CyclicLogic()</c>.  Alternatively, the contents of this method could be reimplemented entirely in which case a call to this method would not be necessary.
VAR
	Result : BOOL;
END_VAR

VAR_INST
	MoverSetPos	 : MoverVector;
	ModXPos		 : LREAL;
	ModXPosRound : LREAL;
	ModYPos		 : LREAL;
	ModYPosRound : LREAL;
	FracX		 : LREAL;
	FracY		 : LREAL;
END_VAR
IF NOT _InitComplete THEN
	_InitComplete := Initialize();
END_IF

//Keep Task command feedbacks up to date
EnableMover.Update();
DisableMover.Update();
HaltMover.Update();
JoinMoverToTrack.Update();
LeaveMoverFromTrack.Update();
ResetMover.Update();
MoveOnTrackXY.Update();
MoveOnTrack.Update();
RotateMover.Update();
ZMove.Update();
AMove.Update();
BMove.Update();
MoveToPosition.Update();
AddMoverToGroup.Update();
JoinToClosestTrack.Update();
SquareMover.Update();
RunExternalSetpointRelativeMode.Update();
StopExternalSetpoint.Update();
EnterMvmtAreaTask.Update();
LeaveMvmtAreaTask.Update();

//Update Mover MC Info
_std	 := _Mover.MCTOPLC.STD;
_Busy	 := _std.Busy.busyMover;
_Error	 := _Mover.Error;
_ErrorID := _Mover.ErrorId;

//Calculate Mover Closest Quarter Angle
_MoverActPos := _Mover.MCTOPLC.ACT.ActPos;
_ModuloPosC	 := MODABS(_MoverActPos.c, 360.0);
IF _ModuloPosC < 315.0 AND _ModuloPosC > 225.0 THEN
	_ClosestQuarterAngle := 270.0;
ELSIF _ModuloPosC < 225.0 AND _ModuloPosC > 135.0 THEN
	_ClosestQuarterAngle := 180.0;
ELSIF _ModuloPosC < 135.0 AND _ModuloPosC > 45.0 THEN
	_ClosestQuarterAngle := 90.0;
ELSE
	_ClosestQuarterAngle := 0.0;
END_IF

//Determine if Mover is at a valid rotation position
MoverSetPos			:= _Mover.MCTOPLC.SET.SetPos;
ModXPos				:= LMOD(MoverSetPos.x, 120.0);
ModXPosRound		:= TO_LREAL(TO_DINT(ModXPos * (2 * 10))) / (2 * 10); //Round the Modulo position to 2 decimal places
FracX				:= FRAC(ModXPosRound);
ModYPos				:= LMOD(MoverSetPos.y, 120.0);
ModYPosRound		:= TO_LREAL(TO_DINT(ModYPos * (2 * 10))) / (2 * 10); //Round the Modulo position to 2 decimal places
FracY				:= FRAC(ModYPosRound);
_AtRotationPosition := (MoverSetPos.x >= 119.8 AND FracX = 0) AND (MoverSetPos.y >= 119.8 AND FracY = 0);

//Monitor Changes in move dynamic settings
IF UpdateMoveDynamics THEN
	_DynMove.SetValuesVADJ(_MoveDynamics.Velocity,
						   _MoveDynamics.Accel,
						   _MoveDynamics.Decel,
						   _MoveDynamics.Jerk);

	_DynTrackMove.SetValuesVADJ(_MoveDynamics.Velocity,
								_MoveDynamics.Accel,
								_MoveDynamics.Decel,
								_MoveDynamics.Jerk);

	UpdateMoveDynamics := FALSE;
END_IF

IF UpdateRotateDynamics THEN
	_DynRotate.SetLimit(Coord_Mcs_C1,
						_RotateDynamics.Velocity,
						_RotateDynamics.Accel,
						_RotateDynamics.Decel,
						_RotateDynamics.Jerk);

	UpdateRotateDynamics := FALSE;
END_IF

IF UpdateTiltDynamics THEN
	_DynRotate.SetLimit(Coord_Mcs_A1,
						_TiltDynamics.Velocity,
						_TiltDynamics.Accel,
						_TiltDynamics.Decel,
						_TiltDynamics.Jerk);

	_DynRotate.SetLimit(Coord_Mcs_B1,
						_TiltDynamics.Velocity,
						_TiltDynamics.Accel,
						_TiltDynamics.Decel,
						_TiltDynamics.Jerk);

	UpdateTiltDynamics := FALSE;
END_IF

//Update Mover Position for HMI
IF _MoverIndex > 0 AND _MoverIndex <= SystemParameters.MOVER_COUNT THEN
	XPlanarHMI.MoverPositions[_MoverIndex] := _MoverActPos;
END_IF
END_METHOD

METHOD Initialize : BOOL
//Set Halt Dynamics
_DynHalt.SetLimit(Coord_Mcs_X, 500.0, 10000.0, 10000.0, 100000.0);
_DynHalt.SetLimit(Coord_Mcs_Y, 500.0, 10000.0, 10000.0, 100000.0);
_DynHalt.SetLimit(Coord_Mcs_Z, 500.0, 10000.0, 10000.0, 100000.0);
_DynHalt.SetLimit(Coord_Mcs_A1, 10.0, 100.0, 100.0, 100.0);
_DynHalt.SetLimit(Coord_Mcs_B1, 10.0, 100.0, 100.0, 100.0);
_DynHalt.SetLimit(Coord_Mcs_C1, 36.0, 360.0, 360.0, 360.0);

IF ipMoverTcIo <> 0 THEN
	_MoverBTN := ipMoverTcIo.GetBtn();
END_IF



(*
HaltDynamics.Mode				  := E_HaltDynamicsMode.AxisX_AxisY_CoordinatedOnPath;
HaltDynamics.PathXY.fVelocity     := 500.0;
HaltDynamics.PathXY.fAcceleration := 10000.0;
HaltDynamics.PathXY.fDeceleration := 10000.0;
HaltDynamics.PathXY.fJerk         := 100000.0;
HaltDynamics.AxisX.fVelocity      := 500.0;
HaltDynamics.AxisX.fAcceleration  := 10000.0;
HaltDynamics.AxisX.fDeceleration  := 10000.0;
HaltDynamics.AxisX.fJerk          := 100000.0;
HaltDynamics.AxisY.fVelocity      := 500.0;
HaltDynamics.AxisY.fAcceleration  := 10000.0;
HaltDynamics.AxisY.fDeceleration  := 10000.0;
HaltDynamics.AxisY.fJerk          := 100000.0;
HaltDynamics.AxisZ.fVelocity      := 500.0;
HaltDynamics.AxisZ.fAcceleration  := 10000.0;
HaltDynamics.AxisZ.fDeceleration  := 10000.0;
HaltDynamics.AxisZ.fJerk          := 100000.0;
HaltDynamics.AxisA.fVelocity      := 10.0;
HaltDynamics.AxisA.fAcceleration  := 100.0;
HaltDynamics.AxisA.fDeceleration  := 100.0;
HaltDynamics.AxisA.fJerk          := 100.0;
HaltDynamics.AxisB.fVelocity      := 10.0;
HaltDynamics.AxisB.fAcceleration  := 100.0;
HaltDynamics.AxisB.fDeceleration  := 100.0;
HaltDynamics.AxisB.fJerk          := 100.0;
HaltDynamics.AxisC.fVelocity      := 36.0;
HaltDynamics.AxisC.fAcceleration  := 360.0;
HaltDynamics.AxisC.fDeceleration  := 360.0;
HaltDynamics.AxisC.fJerk          := 360.0;
*)
END_METHOD

END_FUNCTION_BLOCK

// Part/Tasks/FB_AllowEnable
FUNCTION_BLOCK FB_AllowEnable EXTENDS FB_PartTaskResult
VAR
END_VAR

METHOD Execute : I_PlanarTaskResult
VAR_INPUT
END_VAR
IF NOT HasRun THEN
	_Done	 := FALSE;
	_Error	 := FALSE;
	_Busy	 := FALSE;
	_ErrorID := 0;
	ipPart.pm.AllowEnable(_PlanarFb);
	HasRun := TRUE;
END_IF

Execute := THIS^;
END_METHOD

END_FUNCTION_BLOCK

// XPlanarResultClasses/FB_PartTaskResult
{attribute 'no_explicit_call' := 'do not call this POU directly'}
FUNCTION_BLOCK FB_PartTaskResult EXTENDS FB_PlanarFeedbackResult
VAR
	ipPart : I_XplanarPart;
END_VAR

PROPERTY Part : I_XPlanarPart
SET
ipPart := Part;
END_SET
END_PROPERTY

END_FUNCTION_BLOCK

// Part/I_XPlanarPart
INTERFACE I_XPlanarPart EXTENDS I_BaseFB

METHOD ForceDisable : I_PlanarTaskResult
END_METHOD

PROPERTY ObjectID : OTCID
GET
END_GET
END_PROPERTY

{attribute 'suppress_wrn_C0410'}
PROPERTY pm : REFERENCE TO MC_PlanarPart
GET
END_GET
END_PROPERTY

METHOD Reset : I_PlanarTaskResult
VAR_INPUT
END_VAR
END_METHOD

METHOD SetAllowEnable : I_PlanarTaskResult
END_METHOD

{attribute 'suppress_wrn_C0410'}
PROPERTY State : REFERENCE TO MC_PLANAR_STATE
GET
END_GET
END_PROPERTY

END_INTERFACE

// Part/Tasks/FB_ForceDisable
FUNCTION_BLOCK FB_ForceDisable EXTENDS FB_PartTaskResult
VAR
END_VAR

METHOD Execute : I_PlanarTaskResult
VAR_INPUT
END_VAR
IF NOT HasRun THEN
	_Done	 := FALSE;
	_Error	 := FALSE;
	_Busy	 := FALSE;
	_ErrorID := 0;
	ipPart.pm.ForceDisable(_PlanarFb);
	HasRun := TRUE;
END_IF

Execute := THIS^;
END_METHOD

END_FUNCTION_BLOCK

// Part/Tasks/FB_Initialize
FUNCTION_BLOCK FB_Initialize EXTENDS FB_PartTaskResult
VAR
END_VAR

METHOD Execute : I_PlanarTaskResult
VAR_INPUT
	OID : OTCID;
END_VAR
IF NOT HasRun THEN
	ipPart.pm.Initialize(_PlanarFb, OID, XPlanar.Environment);
	HasRun := TRUE;
END_IF

Execute := THIS^;
END_METHOD

END_FUNCTION_BLOCK

// Part/Tasks/FB_ResetPart
FUNCTION_BLOCK FB_ResetPart EXTENDS FB_PartTaskResult
VAR
END_VAR

METHOD Execute : I_PlanarTaskResult
VAR_INPUT
END_VAR
IF NOT HasRun THEN
	_Done	 := FALSE;
	_Error	 := FALSE;
	_Busy	 := FALSE;
	_ErrorID := 0;
	ipPart.pm.Reset(_PlanarFb);
	HasRun := TRUE;
END_IF

Execute := THIS^;
END_METHOD

END_FUNCTION_BLOCK

// Part/FB_XPlanarPart
{attribute 'no_assign'}
{attribute 'no_explicit_call' := 'do not call this POU directly'}
FUNCTION_BLOCK FB_XPlanarPart EXTENDS FB_CyclicFB IMPLEMENTS I_XPlanarPart
VAR
	{attribute 'suppress_wrn_C0540'}
	PlanarPart			 : MC_PlanarPart;
	_ObjectID			 : OTCID;
	InitPart			 : FB_Initialize   := (Part := THIS^);
	AllowPartEnable		 : FB_AllowEnable  := (Part := THIS^);
	ForcePartDisable	 : FB_ForceDisable := (Part := THIS^);
	ResetPart			 : FB_ResetPart	   := (Part := THIS^);
	InvalidCommandResult : FB_ResultBase   := (Busy := FALSE, Error := TRUE, ErrorID := 9999);
END_VAR

METHOD PUBLIC CyclicLogic
VAR_INPUT
END_VAR
InitPart.Update();
AllowPartEnable.Update();
ForcePartDisable.Update();
ResetPart.Update();
END_METHOD

METHOD ForceDisable : I_PlanarTaskResult
ForceDisable := ForcePartDisable.Execute();
END_METHOD

METHOD Initialize : I_PlanarTaskResult
VAR_INPUT
END_VAR
IF _ObjectID <> 0 THEN
	Initialize := InitPart.Execute(_ObjectID);
ELSE
	Initialize := InvalidCommandResult;
END_IF
END_METHOD

PROPERTY ObjectID : OTCID
GET
ObjectID := _ObjectID;
END_GET
SET
_ObjectID := ObjectID;
END_SET
END_PROPERTY

{attribute 'suppress_wrn_C0410'}
PROPERTY pm : REFERENCE TO MC_PlanarPart
GET
pm  ref= PlanarPart;
END_GET
END_PROPERTY

METHOD Reset : I_PlanarTaskResult
VAR_INPUT
END_VAR
Reset := ResetPart.Execute();
END_METHOD

METHOD SetAllowEnable : I_PlanarTaskResult
SetAllowEnable := AllowPartEnable.Execute();
END_METHOD

{attribute 'suppress_wrn_C0410'}
PROPERTY State : REFERENCE TO MC_PLANAR_STATE
GET
State := PlanarPart.State;
END_GET
END_PROPERTY

END_FUNCTION_BLOCK

// Station/FB_XPlanarStationBase
{attribute 'no_assign_warning'} 
{attribute 'no_explicit_call' := 'do not call this POU directly'}
FUNCTION_BLOCK FB_XPlanarStationBase EXTENDS FB_ComponentBase IMPLEMENTS I_XPlanarStation
VAR
	_Position			 : PositionXYC; //Position of center of the zone
	ipCurrentMover		 : I_XPlanarMover;
	_MoverQueue			 : FB_MoverQueue;
	_NumMoversRequired	 : UDINT := 1;
	_ID					 : UDINT;
	_Size				 : Position2D_LREAL := (x := 120, y := 120); //Size of zone in mm
	_HasMover			 : BOOL;
	_Occupied			 : BOOL;
	ipTrackID			 : UDINT;		 //ID of track that zone resides on
	_CanReleaseMover	 : BOOL := TRUE; //Set to 0 if station area is blocked
	_StationReady AT %Q* : BOOL;
	ipNextStation		 : I_XPlanarStation;
	_AllowQueing		 : BOOL := TRUE;
	_StationComplete	 : BOOL;
	_StationType		 : E_StationType := E_StationType.Process;
	PrepState			 : UDINT;
	StationState		 : E_XplanarStationState;
	_i					 : UDINT := 1;
	_Result 			 : I_PlanarTaskResult;
END_VAR

PROPERTY AllowQueing : BOOL
GET
AllowQueing := _AllowQueing;
END_GET
SET
_AllowQueing := AllowQueing;
END_SET
END_PROPERTY

PROPERTY CanReleaseMover : BOOL
SET
_CanReleaseMover := CanReleaseMover;
END_SET
END_PROPERTY

PROPERTY CurrentMover : I_XPlanarMover
GET
IF ipCurrentMover <> 0 THEN
	CurrentMover := ipCurrentMover;
END_IF
END_GET
END_PROPERTY

PROPERTY Error : BOOL
GET
Error := _Error;
END_GET
END_PROPERTY

METHOD Execute
WatchForMover();
IF ipCurrentMover <> 0 THEN
	CASE StationState OF
		E_XplanarStationState.StationIdle: //Wait for mover to arrive in position
			IF _HasMover AND _StationReady AND NOT _StationComplete THEN
				IF ipCurrentMover <> 0 THEN
					IF (ipTrackID <> 0 AND (ipCurrentMover.Status.CommandMode = MC_PLANAR_MOVER_COMMAND_MODE.OnTrack OR ipCurrentMover.Status.CommandMode = MC_PLANAR_MOVER_COMMAND_MODE.CRotationOnTrack)) OR (ipTrackID = 0 AND (ipCurrentMover.Status.CommandMode = MC_PLANAR_MOVER_COMMAND_MODE.FreeMovement OR ipCurrentMover.Status.CommandMode = MC_PLANAR_MOVER_COMMAND_MODE.CRotationFreeMovement))
						THEN
						StationState := E_XplanarStationState.ProcessMover;
					END_IF
				END_IF
			END_IF

		E_XplanarStationState.ProcessMover: //Perform the desired processes with the mover
			IF _StationComplete THEN
				IF _StationType = E_StationType.MultiMover THEN
					_i			 := 1;
					StationState := E_XPlanarStationState.SendQueue;
				ELSE
					StationState := E_XplanarStationState.SquareUpMover;
				END_IF
			END_IF

		E_XplanarStationState.SquareUpMover: //Check mover for angle that allows X/Y Movement
			IF (ipCurrentMover.Status.CommandMode = MC_PLANAR_MOVER_COMMAND_MODE.CRotationOnTrack) OR (ipCurrentMover.Status.CommandMode = MC_PLANAR_MOVER_COMMAND_MODE.CRotationFreeMovement) THEN
				_Result := ipCurrentMover.MoveCommand.SquareUp();
				IF _Result.Done THEN
					StationState := E_XplanarStationState.SendMoverAway;
				END_IF
			ELSE
				StationState := E_XplanarStationState.SendMoverAway;
			END_IF

		E_XplanarStationState.SendMoverAway: //Send the current lead mover away
			IF ipNextStation <> 0 AND _CanReleaseMover THEN
				IF (NOT ipNextStation.HasMover OR ipNextStation.AllowQueing) THEN
					_Result := ipCurrentMover.MoveCommand.SendToStation(Destination := ipNextStation);
					IF _Result.Busy THEN
						_MoverQueue.Dequeue();
						StationState := E_XplanarStationState.CycleComplete;
					END_IF
				END_IF
			END_IF

		E_XPlanarStationState.SendQueue: //Send the mover queue away
			IF _i <= _NumMoversRequired THEN
				IF _MoverQueue.Queue[1].Destination <> 0 AND _MoverQueue.Queue[1].Destination.ID <> _ID THEN
					_Result := MoverQueue.Queue[1].MoveCommand.SendToStation(Destination := _MoverQueue.Queue[1].Destination);
					IF _Result.Busy THEN
						_MoverQueue.Dequeue();
						_i := _i + 1;
					END_IF
				ELSE
					_Result := MoverQueue.Queue[1].MoveCommand.SendToStation(Destination := ipNextStation);
					IF _Result.Busy THEN
						_MoverQueue.Dequeue();
						_i := _i + 1;
					END_IF
				END_IF
			ELSE
				_i			 := 1;
				StationState := E_XplanarStationState.CycleComplete;
			END_IF

		E_XplanarStationState.CycleComplete: //Mover on its way out
			_StationReady  := FALSE;
			StationState   := E_XplanarStationState.StationIdle;

		E_XPlanarStationState.StationError:
			_Error := TRUE;
	END_CASE
ELSE
	_StationComplete := FALSE;
	_StationReady	 := FALSE;
	StationState	 := E_XplanarStationState.StationIdle;
END_IF
END_METHOD

PROPERTY HasMover : BOOL
GET
HasMover := _HasMover;
END_GET
SET
_HasMover := HasMover;
END_SET
END_PROPERTY

PROPERTY ID : UDINT
GET
ID := _ID;
END_GET
SET
_ID := ID;
END_SET
END_PROPERTY

{attribute 'suppress_wrn_C0410'}
PROPERTY MoverQueue : REFERENCE TO FB_MoverQueue
GET
MoverQueue ref= _MoverQueue;
END_GET
END_PROPERTY

PROPERTY NextStation : I_XPlanarStation
GET
NextStation := ipNextStation;
END_GET
SET
ipNextStation := NextStation;
END_SET
END_PROPERTY

PROPERTY NumMoversRequired : UDINT
GET
NumMoversRequired := _NumMoversRequired;
END_GET
SET
_NumMoversRequired := NumMoversRequired;
END_SET
END_PROPERTY

{attribute 'suppress_wrn_C0410'}
PROPERTY Position : REFERENCE TO PositionXYC
GET
Position ref= _Position;
END_GET
END_PROPERTY

METHOD Reset : BOOL
StationState := E_XplanarStationState.StationIdle;
PrepState	 := 0;
_Error		 := FALSE;
Reset		 := true;
END_METHOD

{attribute 'suppress_wrn_C0410'}
PROPERTY Size : REFERENCE TO Position2D_LREAL
GET
Size ref= _Size;
END_GET
END_PROPERTY

PROPERTY StationComplete : BOOL
SET
_StationComplete := StationComplete;
END_SET
END_PROPERTY

PROPERTY StationReady : BOOL
GET
StationReady := _StationReady;
END_GET
END_PROPERTY

PROPERTY StationType : E_StationType
GET
StationType := _StationType;
END_GET
SET
_StationType := StationType;
END_SET
END_PROPERTY

PROPERTY TrackID : UDINT
GET
TrackID := ipTrackID;
END_GET
SET
ipTrackID := TrackID;
END_SET
END_PROPERTY

METHOD CyclicLogic
VAR
	i : UDINT;
END_VAR
IF _ID > 0 AND _ID <= SystemParameters.STATION_COUNT THEN
	XPlanarHMI.StationObjects[_ID].Width  := TO_DINT(_Size.x);
	XPlanarHMI.StationObjects[_ID].Height := TO_DINT(_Size.y);
	XPlanarHMI.StationObjects[_ID].X	   := TO_DINT(_Position.x);
	XPlanarHMI.StationObjects[_ID].Y	   := TO_DINT(_Position.y);
END_IF

SUPER^.CyclicLogic();
END_METHOD

PROPERTY Name : STRING
GET
Name := _Name;
END_GET
SET
_Name := Name;
END_SET
END_PROPERTY

METHOD WatchForMover
VAR_INST
	idx : UDINT;
END_VAR
FOR idx := 1 TO SystemParameters.MOVER_COUNT DO
	IF ip.Movers[idx] <> 0 THEN
		IF _Position.x > 0 AND _Position.y > 0 THEN
			IF (ip.Movers[idx].ActualPosition.x + SystemParameters.AssumedMoverSize >= _Position.x - (_Size.x / 2) AND ip.Movers[idx].ActualPosition.x - SystemParameters.AssumedMoverSize <= _Position.x + (_Size.x / 2)) AND
			   (ip.Movers[idx].ActualPosition.y + SystemParameters.AssumedMoverSize >= _Position.y - (_Size.y / 2) AND ip.Movers[idx].ActualPosition.y - SystemParameters.AssumedMoverSize <= _Position.y + (_Size.y / 2)) THEN
				IF ip.Movers[idx].Destination <> 0 THEN
					IF ip.Movers[idx].Destination.ID = _ID AND NOT ip.Movers[idx].InStation THEN
						_MoverQueue.Enqueue(ip.Movers[idx]);
						IF SystemParameters.EnableCommandTracing THEN
							Trace(CONCAT(CONCAT('Mover ', TO_STRING(ip.Movers[idx].MoverIndex)), CONCAT(' Queued in station ', TO_STRING(_ID))));
						END_IF
					END_IF
				END_IF
			END_IF
		END_IF
	END_IF
END_FOR

IF _MoverQueue.Count > 0 THEN
	_HasMover	   := TRUE;
	ipCurrentMover := _MoverQueue.FirstMover;
ELSE
	_HasMover	   := FALSE;
	ipCurrentMover := 0;
END_IF

IF _HasMover AND ipCurrentMover <> 0 THEN
	IF ipCurrentMover <> 0 THEN
		CASE _StationType OF
			E_StationType.Process:
				_StationReady := NOT ipCurrentMover.Status.Busy.busyMover;

			E_StationType.MultiMover:
				_StationReady := NOT ipCurrentMover.Status.Busy.busyMover AND (_MoverQueue.Count = _NumMoversRequired);

			E_StationType.DecisionPoint:
				_StationReady := _HasMover;
		END_CASE
	END_IF
END_IF
END_METHOD

END_FUNCTION_BLOCK

// Tile/FB_XPlanarTile
{attribute 'no_assign'}
{attribute 'no_explicit_call' := 'do not call this POU directly'}
FUNCTION_BLOCK FB_XPlanarTile EXTENDS FB_CyclicFB
VAR
	ipTileTcIo			: I_TcIoXPlanarTile;
	_Index				: UINT;
	_Part				: UINT := 1;
	_Btn				: STRING(13);
	_DcLinkVoltage		: UINT;
	_DcLinkOk			: BOOL;
	_TimeToShutdown		: LREAL;
	_ObservedPower		: LREAL;
	_OverLimitFactor	: LREAL;
	_DiagData			: POINTER TO ST_CoeDriveDiagData;
	_Position			: ST_TcIoTilePositionOnPart;
	_Temperatures		: ST_TileTemperatures;
	_TileType			: TileType;
	CoEUpdateTimer		: TON;
	CriticalUpdateTimer : TON;
	DiagDataResult		: ULINT;
END_VAR

PROPERTY Btn : STRING(13)
GET
Btn := _Btn;
END_GET
END_PROPERTY

METHOD PUBLIC CyclicLogic
VAR_INST
	UpdateTileData : BOOL;
	test   : DINT;
END_VAR
IF XPlanar.OperationMode = Tc3_XPlanarUtility.XPlanarOperationMode.Normal THEN
	IF SystemParameters.TileDiagUpdate > 0 THEN
		CoEUpdateTimer(IN := NOT UpdateTileData, PT := TO_TIME(SystemParameters.TileDiagUpdate) * 1000);
		IF CoEUpdateTimer.Q THEN
			UpdateTileData := TRUE;
		END_IF

		test := SIZEOF(_diagdata);

		//Update the tile diagnostic data
		IF UpdateTileData AND_THEN XPlanar.EnvironmentTcIo.TcIoXpu(1).TcIoTile(_Part, Index).CoE.DiagData.Update() THEN
			_DiagData := XPlanar.EnvironmentTcIo.TcIoXpu(1).TcIoTile(_Part, Index).CoE.DiagData.All;
			_DcLinkOk := XPlanar.EnvironmentTcIo.TcIoXpu(1).TcIoTile(_Part, Index).CoE.DiagData.DcLinkOk;
			UpdateTileData	  := FALSE;
		END_IF

		CriticalUpdateTimer(IN := NOT CriticalUpdateTimer.Q, PT := T#1S);
		IF CriticalUpdateTimer.Q THEN
			_TimeToShutdown	 := XPlanar.EnvironmentTcIo.TcIoXpu(1).TcIoTile(_Part, Index).GetTimeToShutdown();
			_ObservedPower	 := XPlanar.EnvironmentTcIo.TcIoXpu(1).TcIoTile(_Part, Index).GetObservedTilePower();
			_OverLimitFactor := XPlanar.EnvironmentTcIo.TcIoXpu(1).TcIoTile(_Part, Index).GetPowerOverLimitFactor();
		END_IF
	ELSE
		UpdateTileData := FALSE;
	END_IF
END_IF
END_METHOD

PROPERTY DcLinkOk : BOOL
GET
DcLinkOk := _DcLinkOk;
END_GET
END_PROPERTY

PROPERTY Index : UINT
GET
Index := _Index;
END_GET
SET
_Index := Index;
END_SET
END_PROPERTY

METHOD Initialize : BOOL
//Get the Tile Type
_TileType := XPlanar.EnvironmentTcIo.TcIoXpu(1).TcIoTile(_Part, _Index).GetTileType();

//Get the configured position of the tile
_Position := XPlanar.EnvironmentTcIo.TcIoXpu(1).TcIoTile(_Part, _Index).TilePositionOnPart();

//Update the object array for HMI
XPlanarHMI.TileObjects[_Index].X := _Position.X;
XPlanarHMI.TileObjects[_Index].Y := _Position.Y;

//Get BTN of tile
_Btn := XPlanar.EnvironmentTcIo.TcIoXpu(1).TcIoTile(_Part, _Index).GetBtn();
CASE _TileType OF
	TileType.APS4244_1000_0000:
		//Update the object array for HMI
		XPlanarHMI.TileObjects[_Index].Width  := 320;
		XPlanarHMI.TileObjects[_Index].Height := 320;
		XPlanar.RotationMultiplier			  := 80.0;

	TileType.APS4322_0000_0000:
		//Update the object array for HMI
		XPlanarHMI.TileObjects[_Index].Width  := 240;
		XPlanarHMI.TileObjects[_Index].Height := 240;
		XPlanar.RotationMultiplier			  := 120.0;

		//Get initial diagnostic data
		IF _Part > 0 AND _Index > 0 THEN
			//ipTileTcIo := XPlanar.EnvironmentTcIo.TcIoXpu(1).TcIoTile(_Part, Index).Aps4322;
			IF XPlanar.OperationMode = Tc3_XPlanarUtility.XPlanarOperationMode.Normal THEN
				IF XPlanar.EnvironmentTcIo.TcIoXpu(1).TcIoTile(_Part, _Index).Aps4322.CoE.DiagData.Update() THEN
					_DiagData := XPlanar.EnvironmentTcIo.TcIoXpu(1).TcIoTile(_Part, _Index).Aps4322.CoE.DiagData.All;
				END_IF
			END_IF
		END_IF
END_CASE

Initialize := TRUE;
END_METHOD

PROPERTY PartIndex : UINT
GET
PartIndex := _Part;
END_GET
SET
_Part := PartIndex;
END_SET
END_PROPERTY

{attribute 'suppress_wrn_C0410'}
PROPERTY PositionOnPart : REFERENCE TO ST_TcIoTilePositionOnPart
GET
PositionOnPart ref= _Position;
END_GET
END_PROPERTY

{attribute 'suppress_wrn_C0410'}
PROPERTY Temperatures : REFERENCE TO ST_TileTemperatures
GET
Temperatures ref= _Temperatures;
END_GET
END_PROPERTY

PROPERTY TimeToShutdown : LREAL
GET
TimeToShutdown := _TimeToShutdown;
END_GET
END_PROPERTY

METHOD Update
VAR_INPUT
END_VAR
XPlanar.EnvironmentTcIo.TcIoXpu(1).TcIoTile(_Part, Index).CoE.DiagData.Update();
_DiagData		 := XPlanar.EnvironmentTcIo.TcIoXpu(1).TcIoTile(_Part, Index).CoE.DiagData.All;
_DcLinkOk		 := XPlanar.EnvironmentTcIo.TcIoXpu(1).TcIoTile(_Part, Index).CoE.DiagData.DcLinkOk;
_TimeToShutdown	 := XPlanar.EnvironmentTcIo.TcIoXpu(1).TcIoTile(_Part, Index).GetTimeToShutdown();
_ObservedPower	 := XPlanar.EnvironmentTcIo.TcIoXpu(1).TcIoTile(_Part, Index).GetObservedTilePower();
_OverLimitFactor := XPlanar.EnvironmentTcIo.TcIoXpu(1).TcIoTile(_Part, Index).GetPowerOverLimitFactor();
END_METHOD

PROPERTY Utility : I_TcIoXPlanarTile
GET
IF ipTileTcIo <> 0 THEN
	Utility := ipTileTcIo;
end_if
END_GET
END_PROPERTY

END_FUNCTION_BLOCK

// Tile/I_XPlanarTile
INTERFACE I_XPlanarTile EXTENDS I_BaseFB

PROPERTY Btn : STRING(13)
GET
END_GET
END_PROPERTY

PROPERTY DcLinkOk : BOOL
GET
END_GET
END_PROPERTY

PROPERTY Index : UINT
GET
END_GET
SET
END_SET
END_PROPERTY

PROPERTY PartIndex : UINT
GET
END_GET
SET
END_SET
END_PROPERTY

{attribute 'suppress_wrn_C0410'}
PROPERTY PositionOnPart : REFERENCE TO ST_TcIoTilePositionOnPart
GET
END_GET
END_PROPERTY

{attribute 'suppress_wrn_C0410'}
PROPERTY Temperatures : REFERENCE TO ST_TileTemperatures
GET
END_GET
END_PROPERTY

PROPERTY TimeToShutdown : UDINT
GET
END_GET
END_PROPERTY

METHOD Update
VAR_INPUT
END_VAR
END_METHOD

PROPERTY Utility : I_TcIoXPlanarTile
GET
END_GET
END_PROPERTY

END_INTERFACE

// Track/TaskClasses/FB_AddTrackToGroup
FUNCTION_BLOCK FB_AddTrackToGroup EXTENDS FB_TrackTaskResult
VAR
END_VAR

METHOD Execute : I_PlanarTaskResult
VAR_INPUT
	refGroup : REFERENCE TO MC_PlanarGroup;
END_VAR
_Done	 := FALSE;
_Error	 := FALSE;
_Busy	 := FALSE;
_ErrorID := 0;
ipTrack.pm.AddToGroup(_PlanarFb, refGroup);
Execute := THIS^;

//Heartbeat that the method is active
ExecuteWatchdog := ExecuteWatchdog + 1;
END_METHOD

END_FUNCTION_BLOCK

// XPlanarResultClasses/FB_TrackTaskResult
{attribute 'no_explicit_call' := 'do not call this POU directly'}
FUNCTION_BLOCK FB_TrackTaskResult EXTENDS FB_PlanarFeedbackResult
VAR
	ipTrack	   : I_XPlanarTrack;
END_VAR

PROPERTY Track : I_XplanarTrack
SET
ipTrack := Track;
END_SET
END_PROPERTY

END_FUNCTION_BLOCK

// Track/TaskClasses/FB_AppendLine
{attribute 'no_assign_warning'} 
FUNCTION_BLOCK FB_AppendLine EXTENDS FB_TrackTaskResult
VAR
	StartPoint : PositionXYC;
	EndPoint   : PositionXYC;
END_VAR

METHOD Execute : I_PlanarTaskResult
VAR_INPUT
	StartPointX : LREAL;
	StartPointY : LREAL;
	EndPointX	: LREAL;
	EndPointY	: LREAL;
END_VAR
IF NOT HasRun THEN
	_Done	 := FALSE;
	_Error	 := FALSE;
	_Busy	 := FALSE;
	_ErrorID := 0;
	StartPoint.SetValuesXY(StartPointX, StartPointY);
	EndPoint.SetValuesXY(EndPointX, EndPointY);
	ipTrack.pm.AppendLine(_PlanarFb, StartPoint, EndPoint);
	HasRun := TRUE;
END_IF

Execute := THIS^;

//Heartbeat that the method is active
ExecuteWatchdog := ExecuteWatchdog + 1;
END_METHOD

END_FUNCTION_BLOCK

// Track/TaskClasses/FB_AppendPoint
{attribute 'no_assign_warning'}
FUNCTION_BLOCK FB_AppendPoint EXTENDS FB_TrackTaskResult
VAR
	Position : PositionXYC;
END_VAR

METHOD Execute : I_PlanarTaskResult
VAR_INPUT
	XPoint : LREAL;
	YPoint : LREAL;
END_VAR
IF NOT HasRun THEN
	_Done	 := FALSE;
	_Error	 := FALSE;
	_Busy	 := FALSE;
	_ErrorID := 0;
	Position.SetValuesXY(XPoint, YPoint);
	ipTrack.pm.AppendPosition(_PlanarFb, Position);
	HasRun := TRUE;
END_IF

Execute := THIS^;

//Heartbeat that the method is active
ExecuteWatchdog := ExecuteWatchdog + 1;
END_METHOD

END_FUNCTION_BLOCK

// Track/TaskClasses/FB_BuildTrack
FUNCTION_BLOCK FB_BuildTrack EXTENDS FB_TrackTaskResult
VAR
	BuildTrack	: BOOL;
END_VAR

METHOD Execute : I_PlanarTaskResult
IF NOT HasRun THEN
	_Done	   := FALSE;
	_Error	   := FALSE;
	_Busy	   := FALSE;
	_ErrorID   := 0;
	BuildTrack := TRUE;
	HasRun	   := TRUE;
END_IF

Execute := THIS^;

//Heartbeat that the method is active
ExecuteWatchdog := ExecuteWatchdog + 1;
END_METHOD

METHOD PUBLIC Update
VAR_INST
	WatchdogCheck : UDINT;
	i			  : UDINT := 1;
END_VAR
_PlanarFb.Update();
CASE TaskState OF
	0: //Init
		THIS^._Busy := FALSE;
		IF BuildTrack THEN
			THIS^._Done	   := FALSE;
			THIS^._Error   := FALSE;
			THIS^._ErrorID := 0;
			THIS^._Busy	   := TRUE;
			BuildTrack	   := FALSE;
			i			   := 1;
			TaskState	   := TaskState + 10;
		END_IF

	10: //Set StartFromTrack
		IF ipTrack.Definition.StartFromTrackID > 0 THEN
			ipTrack.pm.StartFromTrack(_PlanarFb, ip.Tracks[ipTrack.Definition.StartFromTrackID].pm);
			TaskState := TaskState + 1;
		ELSE
			TaskState := TaskState + 10;
		END_IF

	11: //Watch Command Feedback
		IF _PlanarFb.Done THEN
			TaskState := 20;
		ELSIF _PlanarFb.Error THEN
			THIS^._Error			  := TRUE;
			THIS^._ErrorID			  := _PlanarFb.ErrorId;
			THIS^._BlockingObjectInfo := _PlanarFb.objectInfo;
			TaskState				  := 0;
		END_IF

	20: //Append Track Objects
		IF ipTrack.Definition.Items[i].StartPoint.x > 0 THEN
			CASE ipTrack.Definition.Items[i].ItemType OF
				Point:
					ipTrack.pm.AppendPosition(_PlanarFb, ipTrack.Definition.Items[i].StartPoint);

				Line:
					IF ipTrack.Definition.Items[i].EndPoint.x > 0 THEN
						ipTrack.pm.AppendLine(_PlanarFb, ipTrack.Definition.Items[i].StartPoint, ipTrack.Definition.Items[i].EndPoint);
					ELSE
						THIS^._Error			  := TRUE;
						THIS^._ErrorID			  := 9999;
						TaskState				  := 0;	
					END_IF					
					
				Circle:
					ipTrack.pm.AppendCircle(_PlanarFb,
									   ipTrack.Definition.Items[i].StartPoint,
									   ipTrack.Definition.Items[i].EndPoint,
									   ipTrack.Definition.Items[i].CenterPoint,
									   ipTrack.Definition.Items[i].CircleClockwise);
			END_CASE

			TaskState := TaskState + 1;
		ELSE
			TaskState := TaskState + 10; //No Object Defined Exit the loop
		END_IF

	21: //Watch Command Feedback
		IF _PlanarFb.Done THEN
			IF i < SystemParameters.MAX_OBJECTS_PER_TRACK THEN
				i		  := i + 1;
				TaskState := 20;
			ELSE
				i		  := 1;
				TaskState := 30;
			END_IF
		ELSIF _PlanarFb.Error THEN
			THIS^._Error			  := TRUE;
			THIS^._ErrorID			  := _PlanarFb.ErrorId;
			THIS^._BlockingObjectInfo := _PlanarFb.objectInfo;
			TaskState				  := 0;
		END_IF

	30: //Set EndAtTrack
		IF ipTrack.Definition.EndAtTrackID > 0 THEN
			ipTrack.pm.EndAtTrack(_PlanarFb, ip.Tracks[ipTrack.Definition.EndAtTrackID].pm);
			TaskState := TaskState + 1;
		ELSIF ipTrack.Definition.CloseLoop THEN
			ipTrack.pm.CloseLoop(_PlanarFb);
			TaskState := TaskState + 1;
		ELSE
			TaskState := TaskState + 10;
		END_IF

	31: //Watch Command Feedback
		IF _PlanarFb.Done THEN
			TaskState := 40;
		ELSIF _PlanarFb.Error THEN
			THIS^._Error			  := TRUE;
			THIS^._ErrorID			  := _PlanarFb.ErrorId;
			THIS^._BlockingObjectInfo := _PlanarFb.objectInfo;
			TaskState				  := 0;
		END_IF

	40: //Build Complete
		THIS^._Done := TRUE;
		TaskState	:= 0;
END_CASE

IF ExecuteWatchdog <> WatchdogCheck THEN
	WatchdogCheck := ExecuteWatchdog;
ELSE
	HasRun			:= FALSE;
	ExecuteWatchdog := 0;
END_IF
END_METHOD

END_FUNCTION_BLOCK

// Track/TaskClasses/FB_ClearSegment
FUNCTION_BLOCK FB_ClearSegment EXTENDS FB_TrackTaskResult
VAR
END_VAR

METHOD Execute : I_PlanarTaskResult
IF NOT HasRun THEN
	_Done	 := FALSE;
	_Error	 := FALSE;
	_Busy	 := FALSE;
	_ErrorID := 0;
	ipTrack.pm.Clear(_PlanarFb);
	HasRun := TRUE;
END_IF

Execute := THIS^;

//Heartbeat that the method is active
ExecuteWatchdog := ExecuteWatchdog + 1;
END_METHOD

END_FUNCTION_BLOCK

// Track/TaskClasses/FB_CloseLoop
FUNCTION_BLOCK FB_CloseLoop EXTENDS FB_TrackTaskResult
VAR
END_VAR

METHOD Execute : I_PlanarTaskResult
IF NOT HasRun THEN
	_Done	 := FALSE;
	_Error	 := FALSE;
	_Busy	 := FALSE;
	_ErrorID := 0;
	ipTrack.pm.CloseLoop(_PlanarFb);
	HasRun := TRUE;
END_IF

Execute := THIS^;

//Heartbeat that the method is active
ExecuteWatchdog := ExecuteWatchdog + 1;
END_METHOD

END_FUNCTION_BLOCK

// Track/TaskClasses/FB_DisableTrack
FUNCTION_BLOCK FB_DisableTrack EXTENDS FB_TrackTaskResult
VAR
END_VAR

METHOD Execute : I_PlanarTaskResult
VAR_INPUT
END_VAR
IF ipTrack.Status.State = Mc_Planar_State.Enabled THEN
	_Done	 := FALSE;
	_Error	 := FALSE;
	_Busy	 := FALSE;
	_ErrorID := 0;
	ipTrack.pm.Disable(_PlanarFb);
END_IF

Execute := THIS^;

//Heartbeat that the method is active
ExecuteWatchdog := ExecuteWatchdog + 1;
END_METHOD

END_FUNCTION_BLOCK

// Track/TaskClasses/FB_EnableTrack
FUNCTION_BLOCK FB_EnableTrack EXTENDS FB_TrackTaskResult
VAR
END_VAR

METHOD Execute : I_PlanarTaskResult
VAR_INPUT
END_VAR
IF ipTrack.Status.State = Mc_Planar_State.Disabled THEN
	_Done	 := FALSE;
	_Error	 := FALSE;
	_Busy	 := FALSE;
	_ErrorID := 0;
	ipTrack.pm.Enable(_PlanarFb);
END_IF

Execute := THIS^;

//Heartbeat that the method is active
ExecuteWatchdog := ExecuteWatchdog + 1;
END_METHOD

END_FUNCTION_BLOCK

// Track/TaskClasses/FB_SetEndAtTrack
FUNCTION_BLOCK FB_SetEndAtTrack EXTENDS FB_TrackTaskResult
VAR
	Options : ST_EndAtTrackAdvancedOptions;
END_VAR

METHOD Execute : I_PlanarTaskResult
VAR_INPUT
	SegmentID : UDINT;
END_VAR
IF NOT HasRun AND (SegmentID > 0 AND SegmentID <= SystemParameters.TRACK_COUNT) THEN
	_Done	 := FALSE;
	_Error	 := FALSE;
	_Busy	 := FALSE;
	_ErrorID := 0;
	ipTrack.pm.EndAtTrack(_PlanarFb, ip.Tracks[SegmentID].pm);
	HasRun := TRUE;
END_IF

Execute := THIS^;

//Heartbeat that the method is active
ExecuteWatchdog := ExecuteWatchdog + 1;
END_METHOD

END_FUNCTION_BLOCK

// Track/TaskClasses/FB_SetStartFromTrack
FUNCTION_BLOCK FB_SetStartFromTrack EXTENDS FB_TrackTaskResult
VAR
	Options : ST_StartFromTrackAdvancedOptions;
END_VAR

METHOD Execute : I_PlanarTaskResult
VAR_INPUT
	SegmentID : UDINT;
END_VAR
IF NOT HasRun AND (SegmentID > 0 AND SegmentID <= SystemParameters.TRACK_COUNT) THEN
	_Done	 := FALSE;
	_Error	 := FALSE;
	_Busy	 := FALSE;
	_ErrorID := 0;
	ipTrack.pm.StartFromTrack(_PlanarFb, ip.Tracks[SegmentID].pm);
	HasRun := TRUE;
END_IF

Execute := THIS^;

//Heartbeat that the method is active
ExecuteWatchdog := ExecuteWatchdog + 1;
END_METHOD

END_FUNCTION_BLOCK

// Track/TaskClasses/FB_TrackReset
FUNCTION_BLOCK FB_TrackReset EXTENDS FB_TrackTaskResult
VAR
END_VAR

METHOD Execute : I_PlanarTaskResult
IF NOT HasRun THEN
	_Done	 := FALSE;
	_Error	 := FALSE;
	_Busy	 := FALSE;
	_ErrorID := 0;
	ipTrack.pm.Reset(_PlanarFb);
	HasRun := TRUE;
END_IF

Execute := THIS^;

//Heartbeat that the method is active
ExecuteWatchdog := ExecuteWatchdog + 1;
END_METHOD

END_FUNCTION_BLOCK

// Track/FB_XPlanarTrackSegment
{attribute 'no_assign'}
{attribute 'no_explicit_call' := 'do not call this POU directly'}
FUNCTION_BLOCK FB_XPlanarTrackSegment EXTENDS FB_CyclicFB IMPLEMENTS I_XPlanarTrack
VAR
	//Planar Track 
	{attribute 'suppress_wrn_C0540'}
	_Track			: MC_PlanarTrack;
	_Definition		: ST_TrackDefinition;
	ipMcPlanarTrack : I_McPlanarTrack;

